	// Only log if tracing is enabled and the system is now initialized
	IF GPL_Base.TRACING_ENABLED AND_THEN GVL_System.RingBufferLog.P_RingBufferStatus.BaseStatus.Initialized THEN
		BaseStatus.LogEntry.Message								:= Message;
		BaseStatus.LogEntry.Severity							:= Severity;
		BaseStatus.LogEntry.RaiseAlarm							:= RaiseAlarm;
		BaseStatus.LogEntry.InstancePath						:= InstancePath;
		BaseStatus.LogEntry.TaskInfo.AdsPort					:= TwinCAT_SystemInfoVarList._TaskInfo[Tc2_System.GETCURTASKINDEXEX()].AdsPort;
		BaseStatus.LogEntry.TaskInfo.CycleCount					:= TwinCAT_SystemInfoVarList._TaskInfo[Tc2_System.GETCURTASKINDEXEX()].CycleCount;
		BaseStatus.LogEntry.TaskInfo.CycleTime					:= TwinCAT_SystemInfoVarList._TaskInfo[Tc2_System.GETCURTASKINDEXEX()].CycleTime;
		BaseStatus.LogEntry.TaskInfo.CycleTimeExceeded			:= TwinCAT_SystemInfoVarList._TaskInfo[Tc2_System.GETCURTASKINDEXEX()].CycleTimeExceeded;
		BaseStatus.LogEntry.TaskInfo.DcTaskTime					:= TwinCAT_SystemInfoVarList._TaskInfo[Tc2_System.GETCURTASKINDEXEX()].DcTaskTime;
		BaseStatus.LogEntry.TaskInfo.FirstCycle					:= TwinCAT_SystemInfoVarList._TaskInfo[Tc2_System.GETCURTASKINDEXEX()].FirstCycle;
//		BaseStatus.LogEntry.TaskInfo.InCallAfterOutputUpdate	:= TwinCAT_SystemInfoVarList._TaskInfo[Tc2_System.GETCURTASKINDEXEX()].InCallAfterOutputUpdate;
		BaseStatus.LogEntry.TaskInfo.LastExecTime				:= TwinCAT_SystemInfoVarList._TaskInfo[Tc2_System.GETCURTASKINDEXEX()].LastExecTime;
		BaseStatus.LogEntry.TaskInfo.ObjId						:= TwinCAT_SystemInfoVarList._TaskInfo[Tc2_System.GETCURTASKINDEXEX()].ObjId;
		BaseStatus.LogEntry.TaskInfo.Priority					:= TwinCAT_SystemInfoVarList._TaskInfo[Tc2_System.GETCURTASKINDEXEX()].Priority;
		BaseStatus.LogEntry.TaskInfo.RTViolation				:= TwinCAT_SystemInfoVarList._TaskInfo[Tc2_System.GETCURTASKINDEXEX()].RTViolation;
		BaseStatus.LogEntry.TaskInfo.TaskName					:= TwinCAT_SystemInfoVarList._TaskInfo[Tc2_System.GETCURTASKINDEXEX()].TaskName;
		GVL_System.RingBufferLog.AddObject(RefObject := BaseStatus.LogEntry);

		// Verify the entry was added successfully
		IF NOT GVL_System.RingBufferLog.P_ObjectWasAdded THEN
			// AddObject failed - buffer may be full or corrupted
			// Cannot use logging system to report this (would cause recursion)
			// Silently fail - the LogDequeue error handling will detect buffer issues
		ELSE
			// Successfully added - clear the flag
			GVL_System.RingBufferLog.ClearStatusFlagAdded();
		END_IF
	END_IF
END_IF

// Clear re-entry guard before exiting
GVL_System.InReentry_Logging := FALSE;
END_METHOD

END_FUNCTION_BLOCK

// Base/I_BaseStatic
INTERFACE I_BaseStatic EXTENDS __SYSTEM.IQueryInterface

PROPERTY Busy : BOOL
GET
END_GET
END_PROPERTY

PROPERTY Error : BOOL
GET
END_GET
END_PROPERTY

PROPERTY ErrorID : UDINT
GET
END_GET
END_PROPERTY

METHOD Initialize : BOOL
VAR_INPUT
END_VAR
END_METHOD

PROPERTY P_BaseConfiguration : REFERENCE TO ST_BaseConfiguration
GET
END_GET
END_PROPERTY

PROPERTY P_BaseStatus : REFERENCE TO ST_BaseStatus
GET
END_GET
END_PROPERTY

METHOD TraceWithSeverity
VAR_INPUT
	Message		: T_MaxString;
	Severity	: Global.TcEventSeverity;
	RaiseAlarm	: BOOL := FALSE;
END_VAR
END_METHOD

END_INTERFACE

// Base/I_BaseCyclic
INTERFACE I_BaseCyclic EXTENDS I_BaseStatic

METHOD CyclicLogic
END_METHOD

PROPERTY Initialized : BOOL
GET
END_GET
END_PROPERTY

END_INTERFACE

// Command/ITFs/I_Command
INTERFACE I_Command EXTENDS I_BaseCyclic

METHOD Abort : I_Command
END_METHOD

METHOD Cancel : I_Command
END_METHOD

METHOD Complete : I_Command
END_METHOD

METHOD Execute : I_Command
END_METHOD

METHOD InjectConfigurations
VAR_INPUT
    iComponent					: I_ComponentFull;
    iCommandConfiguration 		: I_CommandConfiguration;
    iPermIntlkConfiguration   	: I_PermIntlkConfiguration;
END_VAR
END_METHOD

PROPERTY P_CommandStatus : REFERENCE TO ST_CommandStatus
GET
END_GET
END_PROPERTY

METHOD Pause : I_Command
END_METHOD

METHOD Queue : I_Command
END_METHOD

METHOD Reset : I_Command
END_METHOD

METHOD Resume : I_Command
END_METHOD

METHOD Validate : I_Command
END_METHOD

END_INTERFACE

// Component/ITFs/I_ComponentFull
INTERFACE I_ComponentFull EXTENDS I_ComponentBase

METHOD DequeueCommand : BOOL
VAR_INPUT
	CmdIndex	: DINT;
END_VAR
END_METHOD

METHOD EnqueueCommand
VAR_INPUT
	CmdIndex	: DINT;
END_VAR
END_METHOD

{warning 'Add method implementation or delete method to use base implementation'}
METHOD ExecuteCommand : I_ComponentFull
VAR_INPUT
	CmdIndex	: DINT;
END_VAR
END_METHOD

METHOD PUBLIC GetIndexByPOUName : UINT
VAR_INPUT
	NameIn : T_MaxString;
END_VAR
END_METHOD

{warning 'Add method implementation or delete method to use base implementation'}
METHOD HMICommunication
END_METHOD

METHOD InjectCommandQueue
VAR_INPUT
	iCommandQueue : I_RingBufferICmd;
END_VAR
END_METHOD

PROPERTY P_CommandQueue : I_RingBufferICmd
GET
END_GET
END_PROPERTY

{warning 'Add property implementation or delete property to use base implementation'}
PROPERTY P_ComponentConfiguration : REFERENCE TO ST_ComponentConfiguration
GET
END_GET
END_PROPERTY

{warning 'Add property implementation or delete property to use base implementation'}
PROPERTY P_ComponentStatus : REFERENCE TO ST_ComponentStatus
GET
END_GET
END_PROPERTY

METHOD ResetAllCommands : E_CommandResult
END_METHOD

END_INTERFACE

// Component/ITFs/I_ComponentBase
INTERFACE I_ComponentBase EXTENDS I_BaseCyclic

METHOD InjectSystemInterfaces
VAR_INPUT
	SystemPermIntlk				: I_PermIntlk;
	ControlMode					: I_ControlMode;
END_VAR
END_METHOD

METHOD Reset : E_CommandResult
END_METHOD

END_INTERFACE

// PermIntlk/ITFs/I_PermIntlk
INTERFACE I_PermIntlk EXTENDS I_BaseCyclic

METHOD Evaluate : I_PermIntlk
END_METHOD

METHOD InjectPermIntlkConfiguration
VAR_INPUT
    iPermIntlkCfg 	: I_PermIntlkConfiguration;
END_VAR
END_METHOD

{attribute 'monitoring' := 'call'}
PROPERTY P_OK : BOOL
GET
END_GET
END_PROPERTY

PROPERTY P_PermIntlkStatus : REFERENCE TO ST_PermIntlkStatus
GET
END_GET
END_PROPERTY

END_INTERFACE

// PermIntlk/ITFs/I_PermIntlkConfiguration
INTERFACE I_PermIntlkConfiguration EXTENDS I_BaseStatic

PROPERTY P_PermIntlkConfiguration : REFERENCE TO ST_PermIntlkConfiguration
GET
END_GET
END_PROPERTY

END_INTERFACE

// ControlMode/ITFs/I_ControlMode
INTERFACE I_ControlMode EXTENDS I_BaseCyclic

METHOD ChangeMode : I_ControlMode
VAR_INPUT
	DesiredMode	: DINT;
END_VAR
END_METHOD

PROPERTY P_ControlMode : DINT
GET
END_GET
END_PROPERTY

END_INTERFACE

// RingBuffer/ITFs/I_RingBufferICmd
INTERFACE I_RingBufferICmd EXTENDS I_RingBufferBase

METHOD PUBLIC AddObject
VAR_INPUT
  RefObject           : REFERENCE TO ST_SystimeICmd;
END_VAR
VAR_OUTPUT
  Error               : BOOL;
END_VAR
END_METHOD

PROPERTY P_Buffer : REFERENCE TO ARRAY[GPL_RingBuffer.MIN_NUMBER_OBJECTS..GPL_RingBuffer.MAX_NUMBER_OBJECTS] OF ST_SystimeICmd;
GET
END_GET
END_PROPERTY

PROPERTY P_LastObjectPeeked : REFERENCE TO ST_SystimeICmd
GET
END_GET
END_PROPERTY

PROPERTY P_LastObjectRead : REFERENCE TO ST_SystimeICmd
GET
END_GET
END_PROPERTY

PROPERTY P_LastObjectRemoved : REFERENCE TO ST_SystimeICmd
GET
END_GET
END_PROPERTY

METHOD PUBLIC PeekObject : ST_SystimeICmd
END_METHOD

METHOD PUBLIC ReadObject : ST_SystimeICmd
VAR_OUTPUT
  Error : BOOL;
END_VAR
END_METHOD

END_INTERFACE

// RingBuffer/ITFs/I_RingBufferBase
INTERFACE I_RingBufferBase EXTENDS I_BaseStatic

METHOD ClearLastRemoved
END_METHOD

METHOD ClearStatusFlagAdded
END_METHOD

METHOD ClearStatusFlagPeeked
END_METHOD

METHOD ClearStatusFlagRead
END_METHOD

METHOD ClearStatusFlagRemoved
END_METHOD

PROPERTY P_ObjectWasAdded : REFERENCE TO BOOL
GET
END_GET
END_PROPERTY

PROPERTY P_ObjectWasPeeked : REFERENCE TO BOOL
GET
END_GET
END_PROPERTY

PROPERTY P_ObjectWasRead : REFERENCE TO BOOL
GET
END_GET
END_PROPERTY

PROPERTY P_ObjectWasRemoved : REFERENCE TO BOOL
GET
END_GET
END_PROPERTY

PROPERTY P_RingBufferStatus : REFERENCE TO ST_RingBufferStatus
GET
END_GET
END_PROPERTY

METHOD PUBLIC RemoveObject
VAR_OUTPUT
  Error              : BOOL;
END_VAR
END_METHOD

END_INTERFACE

// Command/ITFs/I_CommandConfiguration
INTERFACE I_CommandConfiguration EXTENDS I_BaseStatic

PROPERTY P_CommandConfiguration : REFERENCE TO ST_CommandConfiguration
GET
END_GET
END_PROPERTY

END_INTERFACE

// Command/ITFs/I_TestClock
INTERFACE I_TestClock

METHOD SetElapsedTime
VAR_INPUT
	DesiredET : LTIME;
END_VAR
END_METHOD

END_INTERFACE

// Command/ITFs/I_Timer
INTERFACE I_Timer EXTENDS __SYSTEM.IQueryInterface

PROPERTY P_ElapsedTime : TIME
GET
END_GET
END_PROPERTY

PROPERTY P_IsElapsed : BOOL
GET
END_GET
END_PROPERTY

METHOD ResetTimer
VAR_INPUT
END_VAR
END_METHOD

METHOD StartTimer
VAR_INPUT
END_VAR
END_METHOD

METHOD StopTimer
VAR_INPUT
END_VAR
END_METHOD

END_INTERFACE

// Command/POUs/FB_Command
{attribute 'no_explicit_call' := 'do not call this POU directly'}
{attribute 'enable_dynamic_creation'}
FUNCTION_BLOCK FB_Command EXTENDS FB_BaseCyclic IMPLEMENTS I_Command, I_CommandConfiguration
VAR
	iCommandInternal			: I_Command := THIS^;
	
 	_iComponent					: I_ComponentFull; // External Dependency
	_iCommandConfiguration		: I_CommandConfiguration; // External Dependency
	_iPermIntlkConfiguration	: I_PermIntlkConfiguration; // External Dependency
	
	LocalCommandConfiguration	: ST_CommandConfiguration := (CommandDescription := 'Missing Command Configuration Interface Reference'); //Local Reference Fallback
	LocalPermIntlkConfiguration	: ST_PermIntlkConfiguration; //Local Reference Fallback

 	fbPermIntlk					: FB_PermIntlkCommand;
	iPermIntlk					: I_PermIntlk := fbPermIntlk;
	
	fbCmdElapsedTime			: FB_CommandElapsedTimer;
	iTimer						: I_Timer := fbCmdElapsedTime;
	
	CommandStatus				: ST_CommandStatus;
	PreviousCommandStatus		: ST_CommandStatus;

	// Auto-reset timing for test compatibility
	CompleteStateCycles						: DINT := 0;
END_VAR

METHOD Abort : I_Command
// Guard condition derived from truth table
// B AND (E OR TO OR (PIC AND AID AND NOT ILK))
// Check external dependencies - only component required for queue operations
// Other dependencies are optional for basic abortion
IF (_iComponent = 0) THEN
	// Only log warning if we have a valid command configuration to read logging settings from
	IF (_iCommandConfiguration <> 0) THEN
		IF __ISVALIDREF(_iCommandConfiguration.P_CommandConfiguration.BaseConfiguration) THEN
			IF _iCommandConfiguration.P_CommandConfiguration.BaseConfiguration.LogTraceConfiguration.What.xLogToEventLogger THEN
				TraceWithSeverity(Message := 'Warning: Missing I_Component external dependency in Abort method - queue operations unavailable', Severity := Global.TcEventSeverity.Warning);
			END_IF
		END_IF
	END_IF
END_IF

// Abort should be available for any command that needs to be stopped or is active
IF SUPER^.BaseStatus.Initialized THEN

// Abort behavior depends on current state
CASE CommandStatus.StepState OF
    E_CommandState.Execute, E_CommandState.Monitor:
        // Abort executing or monitoring command
        _AbortCommand();
        IF (_iCommandConfiguration <> 0) THEN
            IF __ISVALIDREF(_iCommandConfiguration.P_CommandConfiguration.BaseConfiguration) THEN
                IF _iCommandConfiguration.P_CommandConfiguration.BaseConfiguration.LogTraceConfiguration.What.xLogToEventLogger THEN
                    TraceWithSeverity(Message := 'Command aborted during execution', Severity := Global.TcEventSeverity.Info);
                END_IF
            END_IF
        ELSE
            // WARNING: Event logging disabled - configuration interface is null
            TraceWithSeverity(Message := 'WARNING: _iCommandConfiguration is null in Abort - command aborted during execution logging disabled', Severity := Global.TcEventSeverity.Warning);
        END_IF

    E_CommandState.Idle:
        // Check if queued (by result) and remove from queue if present
        IF CommandStatus.Result = E_CommandResult.Accepted THEN // Queued commands have Accepted result
            IF _iComponent <> 0 THEN
                _iComponent.P_CommandQueue.PeekObject(); // peek each
                IF iCommandInternal = _iComponent.P_CommandQueue.P_LastObjectPeeked.iCmd THEN
                    _iComponent.P_CommandQueue.RemoveObject(); // find and remove specific instance
                END_IF
            END_IF
            IF (_iCommandConfiguration <> 0) THEN
                IF __ISVALIDREF(_iCommandConfiguration.P_CommandConfiguration.BaseConfiguration) THEN
                    IF _iCommandConfiguration.P_CommandConfiguration.BaseConfiguration.LogTraceConfiguration.What.xLogToEventLogger THEN
                        TraceWithSeverity(Message := 'Queued command aborted and removed from queue', Severity := Global.TcEventSeverity.Info);
                    END_IF
                END_IF
            ELSE
                // WARNING: Event logging disabled - configuration interface is null
                TraceWithSeverity(Message := 'WARNING: _iCommandConfiguration is null in Abort - queued command aborted and removed from queue logging disabled', Severity := Global.TcEventSeverity.Warning);
            END_IF
        ELSE
            IF (_iCommandConfiguration <> 0) THEN
                IF __ISVALIDREF(_iCommandConfiguration.P_CommandConfiguration.BaseConfiguration) THEN
                    IF _iCommandConfiguration.P_CommandConfiguration.BaseConfiguration.LogTraceConfiguration.What.xLogToEventLogger THEN
                        TraceWithSeverity(Message := 'Idle command marked as aborted', Severity := Global.TcEventSeverity.Info);
                    END_IF
                END_IF
            ELSE
                // WARNING: Event logging disabled - configuration interface is null
                TraceWithSeverity(Message := 'WARNING: _iCommandConfiguration is null in Abort - idle command marked as aborted logging disabled', Severity := Global.TcEventSeverity.Warning);
            END_IF
        END_IF
CommandStatus.Result := E_CommandResult.Aborted;

    E_CommandState.Paused:
        // Abort paused command
        _AbortCommand();
		IF (_iCommandConfiguration <> 0) THEN
			IF __ISVALIDREF(_iCommandConfiguration.P_CommandConfiguration.BaseConfiguration) THEN
				IF _iCommandConfiguration.P_CommandConfiguration.BaseConfiguration.LogTraceConfiguration.What.xLogToEventLogger THEN
					TraceWithSeverity(Message := 'Paused command aborted', Severity := Global.TcEventSeverity.Info);
				END_IF
			END_IF
		ELSE
			// WARNING: Event logging disabled - configuration interface is null
			TraceWithSeverity(Message := 'WARNING: _iCommandConfiguration is null in Abort - paused command aborted logging disabled', Severity := Global.TcEventSeverity.Warning);
		END_IF

    E_CommandState.Complete:
        // Policy: Abort-after-complete should not overwrite terminal results
        IF (_iCommandConfiguration <> 0) THEN
            IF __ISVALIDREF(_iCommandConfiguration.P_CommandConfiguration.BaseConfiguration) THEN
                IF _iCommandConfiguration.P_CommandConfiguration.BaseConfiguration.LogTraceConfiguration.What.xLogToEventLogger THEN
                    TraceWithSeverity(Message := 'Abort ignored - completed command preserves terminal result', Severity := Global.TcEventSeverity.Warning);
                END_IF
            END_IF
        ELSE
            // WARNING: Event logging disabled - configuration interface is null
            TraceWithSeverity(Message := 'WARNING: _iCommandConfiguration is null in Abort - abort ignored for completed command logging disabled', Severity := Global.TcEventSeverity.Warning);
        END_IF
        // Do not change CommandStatus.Result to preserve Ok/RequestTimeout/InterlockLost etc.
END_CASE

ELSE
    // FB not initialized - cannot safely abort
    IF (_iCommandConfiguration <> 0) THEN
        IF __ISVALIDREF(_iCommandConfiguration.P_CommandConfiguration.BaseConfiguration) THEN
            IF _iCommandConfiguration.P_CommandConfiguration.BaseConfiguration.LogTraceConfiguration.What.xLogToEventLogger THEN
                TraceWithSeverity(Message := 'Cannot abort - FB_Command not initialized', Severity := Global.TcEventSeverity.Error);
            END_IF
        END_IF
    ELSE
        // WARNING: Event logging disabled - configuration interface is null
        TraceWithSeverity(Message := 'WARNING: _iCommandConfiguration is null in Abort - FB_Command not initialized logging disabled', Severity := Global.TcEventSeverity.Warning);
    END_IF
END_IF

Abort := THIS^;
END_METHOD

METHOD Cancel : I_Command
// Guard condition derived from truth table
// NOT B AND NOT E AND NOT D
// Check external dependencies - only component required for queue operations
// Other dependencies are optional for basic cancellation
IF (_iComponent = 0) THEN
	// Only log warning if we have a valid command configuration to read logging settings from
	IF (_iCommandConfiguration <> 0) THEN
		IF __ISVALIDREF(_iCommandConfiguration.P_CommandConfiguration.BaseConfiguration) THEN
			IF _iCommandConfiguration.P_CommandConfiguration.BaseConfiguration.LogTraceConfiguration.What.xLogToEventLogger THEN
				TraceWithSeverity(Message := 'Warning: Missing I_Component external dependency in Cancel method - queue operations unavailable', Severity := Global.TcEventSeverity.Warning);
			END_IF
		END_IF
	ELSE
		// WARNING: Event logging disabled - configuration interface is null
		TraceWithSeverity(Message := 'WARNING: _iCommandConfiguration is null in Cancel - missing I_Component dependency logging disabled', Severity := Global.TcEventSeverity.Warning);
	END_IF
END_IF

// Cancel behavior depends on current state, not on Done flag
// Allow cancel for idle and paused states regardless of Done status
CASE CommandStatus.StepState OF
    E_CommandState.Idle:
        // Check if queued (by result) and remove from queue if present
        IF CommandStatus.Result = E_CommandResult.Accepted THEN // Queued commands have Accepted result
            IF _iComponent <> 0 THEN
                _iComponent.P_CommandQueue.PeekObject(); // peek each
                IF iCommandInternal = _iComponent.P_CommandQueue.P_LastObjectPeeked.iCmd THEN
                    _iComponent.P_CommandQueue.RemoveObject(); // find and remove specific instance
                END_IF
            END_IF
            IF (_iCommandConfiguration <> 0) THEN
                IF __ISVALIDREF(_iCommandConfiguration.P_CommandConfiguration.BaseConfiguration) THEN
                    IF _iCommandConfiguration.P_CommandConfiguration.BaseConfiguration.LogTraceConfiguration.What.xLogToEventLogger THEN
                        TraceWithSeverity(Message := 'Queued command cancelled and removed from queue', Severity := Global.TcEventSeverity.Info);
                    END_IF
                END_IF
            ELSE
                // WARNING: Event logging disabled - configuration interface is null
                TraceWithSeverity(Message := 'WARNING: _iCommandConfiguration is null in Cancel - queued command cancelled logging disabled', Severity := Global.TcEventSeverity.Warning);
            END_IF
        ELSE
            // Regular idle command - still set cancelled result
            IF (_iCommandConfiguration <> 0) THEN
                IF __ISVALIDREF(_iCommandConfiguration.P_CommandConfiguration.BaseConfiguration) THEN
                    IF _iCommandConfiguration.P_CommandConfiguration.BaseConfiguration.LogTraceConfiguration.What.xLogToEventLogger THEN
                        TraceWithSeverity(Message := 'Idle command cancelled', Severity := Global.TcEventSeverity.Info);
                    END_IF
                END_IF
            ELSE
                // WARNING: Event logging disabled - configuration interface is null
                TraceWithSeverity(Message := 'WARNING: _iCommandConfiguration is null in Cancel - idle command cancelled logging disabled', Severity := Global.TcEventSeverity.Warning);
            END_IF
        END_IF
        // Set cancelled result for any idle command, stay in Idle state
        CommandStatus.Result := E_CommandResult.Cancelled;
                IF __ISVALIDREF(CommandStatus.BaseStatus) THEN
            CommandStatus.BaseStatus.Error := FALSE;  // Cancelled is not an error
                    ELSE
            TraceWithSeverity(Message := 'Command Base Reference Data Structure not present - see _InitializeReferences', Severity := Global.TcEventSeverity.Error);
        END_IF
        
    E_CommandState.Execute, E_CommandState.Monitor:
        // Policy: Cancel should not change results while busy - do nothing
        IF (_iCommandConfiguration <> 0) THEN
            IF __ISVALIDREF(_iCommandConfiguration.P_CommandConfiguration.BaseConfiguration) THEN
                IF _iCommandConfiguration.P_CommandConfiguration.BaseConfiguration.LogTraceConfiguration.What.xLogToEventLogger THEN
                    TraceWithSeverity(Message := 'Cancel rejected - command is executing, use Abort instead', Severity := Global.TcEventSeverity.Warning);
                END_IF
            END_IF
        ELSE
            // WARNING: Event logging disabled - configuration interface is null
            TraceWithSeverity(Message := 'WARNING: _iCommandConfiguration is null in Cancel - cancel rejected (executing) logging disabled', Severity := Global.TcEventSeverity.Warning);
        END_IF
        // Do not change CommandStatus.Result
        
    E_CommandState.Paused:
        // Policy: Cancel should not change results while paused/busy - do nothing
        IF (_iCommandConfiguration <> 0) THEN
            IF __ISVALIDREF(_iCommandConfiguration.P_CommandConfiguration.BaseConfiguration) THEN
                IF _iCommandConfiguration.P_CommandConfiguration.BaseConfiguration.LogTraceConfiguration.What.xLogToEventLogger THEN
                    TraceWithSeverity(Message := 'Cancel rejected - command is paused, use Abort instead', Severity := Global.TcEventSeverity.Warning);
                END_IF
            END_IF
        ELSE
            // WARNING: Event logging disabled - configuration interface is null
            TraceWithSeverity(Message := 'WARNING: _iCommandConfiguration is null in Cancel - cancel rejected (paused) logging disabled', Severity := Global.TcEventSeverity.Warning);
        END_IF
        // Do not change CommandStatus.Result

    E_CommandState.Complete:
        // Policy: Cancel should not change results while complete - do nothing
        IF (_iCommandConfiguration <> 0) THEN
            IF __ISVALIDREF(_iCommandConfiguration.P_CommandConfiguration.BaseConfiguration) THEN
                IF _iCommandConfiguration.P_CommandConfiguration.BaseConfiguration.LogTraceConfiguration.What.xLogToEventLogger THEN
                    TraceWithSeverity(Message := 'Cancel rejected - command is complete', Severity := Global.TcEventSeverity.Warning);
                END_IF
            END_IF
        ELSE
            // WARNING: Event logging disabled - configuration interface is null
            TraceWithSeverity(Message := 'WARNING: _iCommandConfiguration is null in Cancel - cancel rejected (complete) logging disabled', Severity := Global.TcEventSeverity.Warning);
        END_IF
        // Do not change CommandStatus.Result
END_CASE

Cancel := THIS^;
END_METHOD

METHOD Complete : I_Command
// Mark command as no longer busy when completion is triggered
// This allows the component to accept new commands immediately
IF CommandStatus.StepState = E_CommandState.Monitor THEN
    IF __ISVALIDREF(CommandStatus.BaseStatus) THEN
        CommandStatus.BaseStatus.Busy := FALSE;
            ELSE
        TraceWithSeverity(Message := 'Command Base Reference Data Structure not present - see _InitializeReferences', Severity := Global.TcEventSeverity.Error);
    END_IF
    // Stop the elapsed timer to prevent it from continuing to increment
    IF iTimer <> 0 THEN
        iTimer.StopTimer();
    END_IF
END_IF

Complete := THIS^;
END_METHOD

METHOD Execute : I_Command
// Critical check: Timer interface must be present for command execution
IF iTimer = 0 THEN
	TraceWithSeverity(
		Message := 'CRITICAL: Cannot execute command - timer interface not present! Timeout monitoring would not work!',
		Severity := Global.TcEventSeverity.Error
	);
	CommandStatus.Result := E_CommandResult.BadRequest;
	Execute := THIS^;
	RETURN;
END_IF

// Guard condition derived from truth table
// NOT B AND NOT E AND NOT D AND ILK AND NOT TO
// Check external dependencies - allow execution with minimal configuration for basic testing
IF (_iComponent = 0) THEN
	// Only log warning if we have a valid command configuration to read logging settings from
	IF (_iCommandConfiguration <> 0) THEN
		IF __ISVALIDREF(_iCommandConfiguration.P_CommandConfiguration.BaseConfiguration) THEN
			IF _iCommandConfiguration.P_CommandConfiguration.BaseConfiguration.LogTraceConfiguration.What.xLogToEventLogger THEN
				TraceWithSeverity(Message := 'Warning: Missing I_Component external dependency in Execute method - advanced features unavailable', Severity := Global.TcEventSeverity.Warning);
			END_IF
		END_IF
	END_IF
END_IF

// Check timeout condition safely
IF (_iCommandConfiguration <> 0) THEN
    IF CommandStatus.LastCommandElapsedTime >= TIME_TO_LTIME(_iCommandConfiguration.P_CommandConfiguration.TimeoutTime) THEN
        CommandStatus.Result := E_CommandResult.RequestTimeout;
                IF __ISVALIDREF(CommandStatus.BaseStatus) THEN
            CommandStatus.BaseStatus.Error := TRUE;  // Set error flag for timeout
                        CommandStatus.BaseStatus.Done := TRUE;  // Complete state always sets Done=TRUE (terminal state)
                    ELSE
            TraceWithSeverity(Message := 'Command Base Reference Data Structure not present - see _InitializeReferences', Severity := Global.TcEventSeverity.Error);
        END_IF
        IF __ISVALIDREF(_iCommandConfiguration.P_CommandConfiguration.BaseConfiguration) THEN
            IF _iCommandConfiguration.P_CommandConfiguration.BaseConfiguration.LogTraceConfiguration.What.xLogToEventLogger THEN
                TraceWithSeverity(Message := 'Command timeout exceeded in Execute method', Severity := Global.TcEventSeverity.Error);
            END_IF
        END_IF
    END_IF
ELSE
    // WARNING: Cannot check timeout without configuration - execution may proceed beyond timeout
    TraceWithSeverity(Message := 'WARNING: _iCommandConfiguration is null in Execute method - timeout check bypassed', Severity := Global.TcEventSeverity.Warning);
END_IF

// Enhanced guard conditions - prevent execution in terminal states
// Execute should only be allowed from clean Idle state
IF SUPER^.BaseStatus.Initialized AND 
   NOT CommandStatus.BaseStatus.Busy AND 
   NOT CommandStatus.BaseStatus.Done AND
   NOT CommandStatus.BaseStatus.Error THEN

// Execute behavior depends on current state
CASE CommandStatus.StepState OF
    E_CommandState.Idle:
        // Execute must validate before accepting - call Validate() internally
        _ValidateCommand();
        
        // Only proceed if validation was successful (Accepted)
        IF CommandStatus.Result = E_CommandResult.Accepted THEN
            
            // Optional trace
            IF (_iCommandConfiguration <> 0) THEN
                IF __ISVALIDREF(_iCommandConfiguration.P_CommandConfiguration.BaseConfiguration) THEN
                    IF _iCommandConfiguration.P_CommandConfiguration.BaseConfiguration.LogTraceConfiguration.When = E_LogTraceWhen.xRunCyclic AND_THEN
                       _iCommandConfiguration.P_CommandConfiguration.BaseConfiguration.LogTraceConfiguration.What.xLogToEventLogger THEN
                        _LogCommand();
                    END_IF
                END_IF
            ELSE
                // WARNING: Event logging disabled - configuration interface is null
                TraceWithSeverity(Message := 'WARNING: _iCommandConfiguration is null in Execute - optional trace logging disabled', Severity := Global.TcEventSeverity.Warning);
            END_IF
            
            // Set Busy flag to enable state transitions - validation already passed
            IF __ISVALIDREF(CommandStatus.BaseStatus) THEN
                CommandStatus.BaseStatus.Busy := TRUE;
                            ELSE
                TraceWithSeverity(Message := 'Command Base Reference Data Structure not present - see _InitializeReferences', Severity := Global.TcEventSeverity.Error);
            END_IF

            // Start the command timer to track elapsed time
            IF iTimer <> 0 THEN
                iTimer.StartTimer();
            END_IF
            // Keep Result as Accepted - CyclicLogic will drive state progression
        END_IF
        // If validation failed, Result already contains the failure reason (Forbidden, BadRequest, etc.)
        
    E_CommandState.Execute, E_CommandState.Monitor, E_CommandState.Complete:
        // Already executing, monitoring, or complete - cannot execute again
        // Complete is a terminal state - use Reset() to return to Idle for re-execution
        IF (_iCommandConfiguration <> 0) THEN
            IF __ISVALIDREF(_iCommandConfiguration.P_CommandConfiguration.BaseConfiguration) THEN
                IF _iCommandConfiguration.P_CommandConfiguration.BaseConfiguration.LogTraceConfiguration.What.xLogToEventLogger THEN
                    TraceWithSeverity(Message := 'Cannot execute - command already in progress or complete. Use Reset() first.', Severity := Global.TcEventSeverity.Warning);
                END_IF
            END_IF
        ELSE
            // WARNING: Event logging disabled - configuration interface is null
            TraceWithSeverity(Message := 'WARNING: _iCommandConfiguration is null in Execute - already in progress/complete logging disabled', Severity := Global.TcEventSeverity.Warning);
        END_IF

    E_CommandState.Paused:
        // Cannot execute from paused state - use Resume instead
        IF (_iCommandConfiguration <> 0) THEN
            IF __ISVALIDREF(_iCommandConfiguration.P_CommandConfiguration.BaseConfiguration) THEN
                IF _iCommandConfiguration.P_CommandConfiguration.BaseConfiguration.LogTraceConfiguration.What.xLogToEventLogger THEN
                    TraceWithSeverity(Message := 'Cannot execute - command is paused, use Resume instead', Severity := Global.TcEventSeverity.Warning);
                END_IF
            END_IF
        ELSE
            // WARNING: Event logging disabled - configuration interface is null
            TraceWithSeverity(Message := 'WARNING: _iCommandConfiguration is null in Execute - paused state logging disabled', Severity := Global.TcEventSeverity.Warning);
        END_IF
END_CASE

ELSE
	// Guard condition not met - command not initialized, busy, or in terminal state
	IF NOT SUPER^.BaseStatus.Initialized THEN
	    CommandStatus.Result := E_CommandResult.BadRequest;
	    	    IF __ISVALIDREF(CommandStatus.BaseStatus) THEN
	        CommandStatus.BaseStatus.Error := TRUE;  // Set error flag for bad request
	        	    ELSE
	        TraceWithSeverity(Message := 'Command Base Reference Data Structure not present - see _InitializeReferences', Severity := Global.TcEventSeverity.Error);
	    END_IF
	    IF (_iCommandConfiguration <> 0) THEN
	    	IF __ISVALIDREF(_iCommandConfiguration.P_CommandConfiguration.BaseConfiguration) THEN
	            IF _iCommandConfiguration.P_CommandConfiguration.BaseConfiguration.LogTraceConfiguration.What.xLogToEventLogger THEN
	                TraceWithSeverity(Message := 'Execute failed - command not initialized', Severity := Global.TcEventSeverity.Warning);
	            END_IF
	        END_IF
	    ELSE
	        // WARNING: Event logging disabled - configuration interface is null
	        TraceWithSeverity(Message := 'WARNING: _iCommandConfiguration is null in Execute - not initialized logging disabled', Severity := Global.TcEventSeverity.Warning);
	    END_IF
	ELSIF CommandStatus.BaseStatus.Busy THEN
	    CommandStatus.Result := E_CommandResult.Forbidden;
	    	    IF __ISVALIDREF(CommandStatus.BaseStatus) THEN
	        CommandStatus.BaseStatus.Error := TRUE;  // Set error flag for forbidden
	        	    ELSE
	        TraceWithSeverity(Message := 'Command Base Reference Data Structure not present - see _InitializeReferences', Severity := Global.TcEventSeverity.Error);
	    END_IF
	    IF (_iCommandConfiguration <> 0) THEN
	    	IF __ISVALIDREF(_iCommandConfiguration.P_CommandConfiguration.BaseConfiguration) THEN
	            IF _iCommandConfiguration.P_CommandConfiguration.BaseConfiguration.LogTraceConfiguration.What.xLogToEventLogger THEN
	                TraceWithSeverity(Message := 'Execute failed - command busy', Severity := Global.TcEventSeverity.Warning);
	            END_IF
	        END_IF
	    ELSE
	        // WARNING: Event logging disabled - configuration interface is null
	        TraceWithSeverity(Message := 'WARNING: _iCommandConfiguration is null in Execute - command busy logging disabled', Severity := Global.TcEventSeverity.Warning);
	    END_IF
	END_IF
END_IF

Execute := THIS^;
END_METHOD

METHOD InjectConfigurations
VAR_INPUT
    iComponent					: I_ComponentFull;
    iCommandConfiguration 		: I_CommandConfiguration;
    iPermIntlkConfiguration   	: I_PermIntlkConfiguration;
END_VAR
// Inject component interface (moved from FB_Init)
IF iComponent <> 0 THEN
	THIS^._iComponent := iComponent;
	IF NOT SUPER^.BaseStatus.LogTraceStatus.ComponentInterfaceInjectedShown THEN
		TraceWithSeverity(Message := 'FB_Command: Component interface injected successfully', Severity := Global.TcEventSeverity.Verbose);
		SUPER^.BaseStatus.LogTraceStatus.ComponentInterfaceInjectedShown := TRUE;
	END_IF
END_IF

// Inject configuration interfaces (allow null interfaces for testing)
// Null interfaces clear the stored reference to force fallback to local config
IF iCommandConfiguration <> 0 THEN
    _iCommandConfiguration := iCommandConfiguration;
    IF NOT SUPER^.BaseStatus.LogTraceStatus.CmdConfigInterfaceInjectedShown THEN
		TraceWithSeverity(Message := 'FB_Command: Command configuration interface injected successfully', Severity := Global.TcEventSeverity.Verbose);
		SUPER^.BaseStatus.LogTraceStatus.CmdConfigInterfaceInjectedShown := TRUE;
	END_IF
ELSE
    IF (_iCommandConfiguration <> 0) THEN
        IF __ISVALIDREF(_iCommandConfiguration.P_CommandConfiguration.BaseConfiguration) THEN
            IF _iCommandConfiguration.P_CommandConfiguration.BaseConfiguration.LogTraceConfiguration.What.xLogToEventLogger THEN
                TraceWithSeverity(Message := 'Null Command Configuration interface injected - clearing reference', Severity := Global.TcEventSeverity.Info);
            END_IF
        END_IF
    END_IF
    _iCommandConfiguration := 0; // Clear the reference
END_IF

IF iPermIntlkConfiguration <> 0 THEN
    _iPermIntlkConfiguration := iPermIntlkConfiguration;
    IF NOT SUPER^.BaseStatus.LogTraceStatus.PermIntlkConfigInjectedShown THEN
		TraceWithSeverity(Message := 'FB_Command: PermIntlk configuration interface injected successfully', Severity := Global.TcEventSeverity.Verbose);
		SUPER^.BaseStatus.LogTraceStatus.PermIntlkConfigInjectedShown := TRUE;
	END_IF
ELSE
    IF (_iCommandConfiguration <> 0) THEN
        IF __ISVALIDREF(_iCommandConfiguration.P_CommandConfiguration.BaseConfiguration) THEN
            IF _iCommandConfiguration.P_CommandConfiguration.BaseConfiguration.LogTraceConfiguration.What.xLogToEventLogger THEN
                TraceWithSeverity(Message := 'Null PermIntlk Configuration interface injected - clearing reference', Severity := Global.TcEventSeverity.Info);
            END_IF
        END_IF
    END_IF
    _iPermIntlkConfiguration := 0; // Clear the reference
END_IF

// Only inject to child objects if interfaces are valid
IF iCommandConfiguration <> 0 THEN
    fbPermIntlk.InjectCommandConfiguration(iCommandCfg := iCommandConfiguration);
    fbCmdElapsedTime.InjectConfiguration(iCommand := THIS^, iCommandConfiguration := iCommandConfiguration);
    IF NOT SUPER^.BaseStatus.LogTraceStatus.ConfigsInjectedToChildrenShown THEN
		TraceWithSeverity(Message := 'FB_Command: Configurations injected to child objects (fbPermIntlk, fbCmdElapsedTime)', Severity := Global.TcEventSeverity.Verbose);
		SUPER^.BaseStatus.LogTraceStatus.ConfigsInjectedToChildrenShown := TRUE;
	END_IF
END_IF

IF iPermIntlkConfiguration <> 0 THEN
    fbPermIntlk.InjectPermIntlkConfiguration(iPermIntlkCfg := iPermIntlkConfiguration);
    // Ensure permissive interface is properly initialized
    fbPermIntlk.Initialize();
    IF NOT SUPER^.BaseStatus.LogTraceStatus.PermIntlkInitializedShown THEN
		TraceWithSeverity(Message := 'FB_Command: PermIntlk configuration injected and initialized in fbPermIntlk', Severity := Global.TcEventSeverity.Verbose);
		SUPER^.BaseStatus.LogTraceStatus.PermIntlkInitializedShown := TRUE;
	END_IF
END_IF

// Initialize the command after dependency injection
// This ensures all interfaces are available before initialization
THIS^.Initialize();

// Set BadRequest result if required configurations are missing (fail-closed policy)
IF (_iCommandConfiguration = 0) OR (_iPermIntlkConfiguration = 0) THEN
    CommandStatus.Result := E_CommandResult.BadRequest;
        IF __ISVALIDREF(CommandStatus.BaseStatus) THEN
        CommandStatus.BaseStatus.Error := TRUE;
            ELSE
        TraceWithSeverity(Message := 'Command Base Reference Data Structure not present - see _InitializeReferences', Severity := Global.TcEventSeverity.Error);
    END_IF
END_IF;
END_METHOD

PROPERTY P_CommandStatus : REFERENCE TO ST_CommandStatus
GET
P_CommandStatus REF= _ResolveCommandStatus();
END_GET
END_PROPERTY

METHOD Pause : I_Command
// Guard condition derived from truth table
// B AND NOT E AND NOT D
// Check external dependencies - allow basic pause functionality with warnings
IF (_iComponent = 0) THEN
	// Only log warning if we have a valid command configuration to read logging settings from
	IF (_iCommandConfiguration <> 0) THEN
		IF __ISVALIDREF(_iCommandConfiguration.P_CommandConfiguration) THEN
			IF __ISVALIDREF(_iCommandConfiguration.P_CommandConfiguration.BaseConfiguration) THEN
				IF _iCommandConfiguration.P_CommandConfiguration.BaseConfiguration.LogTraceConfiguration.What.xLogToEventLogger THEN
					TraceWithSeverity(Message := 'Warning: Missing I_Component external dependency in Pause method', Severity := Global.TcEventSeverity.Warning);
				END_IF
			END_IF
		END_IF
	ELSE
		// WARNING: Event logging disabled - configuration interface is null
		TraceWithSeverity(Message := 'WARNING: _iCommandConfiguration is null in Pause - missing I_Component dependency logging disabled', Severity := Global.TcEventSeverity.Warning);
	END_IF
END_IF

IF CommandStatus.BaseStatus.Busy AND 
   NOT CommandStatus.BaseStatus.Error AND 
   NOT CommandStatus.BaseStatus.Done THEN

// Pause behavior depends on current state
CASE CommandStatus.StepState OF
    E_CommandState.Execute, E_CommandState.Monitor:
        // Pause executing or monitoring command
        CommandStatus.StepState := E_CommandState.Paused;
                // Keep Busy = TRUE while paused (paused commands are active but suspended)
        // CommandStatus.BaseStatus.Busy remains TRUE
        IF (_iCommandConfiguration <> 0) THEN
            IF __ISVALIDREF(_iCommandConfiguration.P_CommandConfiguration.BaseConfiguration) THEN
                IF _iCommandConfiguration.P_CommandConfiguration.BaseConfiguration.LogTraceConfiguration.What.xLogToEventLogger THEN
                    TraceWithSeverity(Message := 'Command paused during execution', Severity := Global.TcEventSeverity.Info);
                END_IF
            END_IF
        ELSE
            // WARNING: Event logging disabled - configuration interface is null
            TraceWithSeverity(Message := 'WARNING: _iCommandConfiguration is null in Pause - command paused during execution logging disabled', Severity := Global.TcEventSeverity.Warning);
        END_IF
        
    // Note: Queued commands are now Idle with Accepted result
        
    E_CommandState.Idle:
        // Cannot pause idle command
        IF (_iCommandConfiguration <> 0) THEN
            IF __ISVALIDREF(_iCommandConfiguration.P_CommandConfiguration.BaseConfiguration) THEN
                IF _iCommandConfiguration.P_CommandConfiguration.BaseConfiguration.LogTraceConfiguration.What.xLogToEventLogger THEN
                    TraceWithSeverity(Message := 'Cannot pause idle command', Severity := Global.TcEventSeverity.Warning);
                END_IF
            END_IF
        ELSE
            // WARNING: Event logging disabled - configuration interface is null
            TraceWithSeverity(Message := 'WARNING: _iCommandConfiguration is null in Pause - cannot pause idle command logging disabled', Severity := Global.TcEventSeverity.Warning);
        END_IF
        
    E_CommandState.Paused:
        // Already paused
        IF (_iCommandConfiguration <> 0) THEN
            IF __ISVALIDREF(_iCommandConfiguration.P_CommandConfiguration.BaseConfiguration) THEN
                IF _iCommandConfiguration.P_CommandConfiguration.BaseConfiguration.LogTraceConfiguration.What.xLogToEventLogger THEN
                    TraceWithSeverity(Message := 'Command is already paused', Severity := Global.TcEventSeverity.Info);
                END_IF
            END_IF
        ELSE
            // WARNING: Event logging disabled - configuration interface is null
            TraceWithSeverity(Message := 'WARNING: _iCommandConfiguration is null in Pause - already paused logging disabled', Severity := Global.TcEventSeverity.Warning);
        END_IF
        
    E_CommandState.Complete:
        // Cannot pause completed command
        IF (_iCommandConfiguration <> 0) THEN
            IF __ISVALIDREF(_iCommandConfiguration.P_CommandConfiguration.BaseConfiguration) THEN
                IF _iCommandConfiguration.P_CommandConfiguration.BaseConfiguration.LogTraceConfiguration.What.xLogToEventLogger THEN
                    TraceWithSeverity(Message := 'Cannot pause completed command', Severity := Global.TcEventSeverity.Warning);
                END_IF
            END_IF
        ELSE
            // WARNING: Event logging disabled - configuration interface is null
            TraceWithSeverity(Message := 'WARNING: _iCommandConfiguration is null in Pause - cannot pause completed command logging disabled', Severity := Global.TcEventSeverity.Warning);
        END_IF
END_CASE

ELSE
	// Guard condition not met - pause not allowed
	IF (_iCommandConfiguration <> 0) THEN
		IF __ISVALIDREF(_iCommandConfiguration.P_CommandConfiguration.BaseConfiguration) THEN
			IF _iCommandConfiguration.P_CommandConfiguration.BaseConfiguration.LogTraceConfiguration.What.xLogToEventLogger THEN
				TraceWithSeverity(Message := 'Pause guard condition not met', Severity := Global.TcEventSeverity.Warning);
			END_IF
		END_IF
	ELSE
		// WARNING: Event logging disabled - configuration interface is null
		TraceWithSeverity(Message := 'WARNING: _iCommandConfiguration is null in Pause - guard condition not met logging disabled', Severity := Global.TcEventSeverity.Warning);
	END_IF
END_IF

Pause := THIS^;
END_METHOD

METHOD Queue : I_Command
// Guard condition derived from truth table
// NOT B AND NOT E
// Check external dependencies
IF (_iComponent = 0) THEN
	// Only log warning if we have a valid command configuration to read logging settings from
	IF (_iCommandConfiguration <> 0) THEN
		IF __ISVALIDREF(_iCommandConfiguration.P_CommandConfiguration) THEN
			IF __ISVALIDREF(_iCommandConfiguration.P_CommandConfiguration.BaseConfiguration) THEN
				IF _iCommandConfiguration.P_CommandConfiguration.BaseConfiguration.LogTraceConfiguration.What.xLogToEventLogger THEN
					TraceWithSeverity(Message := 'Missing I_Component external dependency in Queue method', Severity := Global.TcEventSeverity.Error);
				END_IF
			END_IF
		END_IF
	ELSE
		// WARNING: Event logging disabled - configuration interface is null
		TraceWithSeverity(Message := 'WARNING: _iCommandConfiguration is null in Queue - missing I_Component dependency logging disabled', Severity := Global.TcEventSeverity.Warning);
	END_IF
	RETURN;
END_IF
IF (_iCommandConfiguration = 0) THEN
	// CRITICAL: Cannot queue without command configuration
	TraceWithSeverity(Message := 'CRITICAL: _iCommandConfiguration is null in Queue method - queue operation rejected', Severity := Global.TcEventSeverity.Error);
	RETURN;
END_IF
IF (_iPermIntlkConfiguration = 0) THEN
	// Log using the valid command configuration we already verified exists
	IF __ISVALIDREF(_iCommandConfiguration.P_CommandConfiguration) THEN
		IF __ISVALIDREF(_iCommandConfiguration.P_CommandConfiguration.BaseConfiguration) THEN
			IF _iCommandConfiguration.P_CommandConfiguration.BaseConfiguration.LogTraceConfiguration.What.xLogToEventLogger THEN
				TraceWithSeverity(Message := 'Missing I_PermIntlkConfiguration external dependency in Queue method', Severity := Global.TcEventSeverity.Error);
			END_IF
		END_IF
	END_IF
	RETURN;
END_IF

IF NOT CommandStatus.BaseStatus.Busy AND 
   NOT CommandStatus.BaseStatus.Error THEN

// Queue behavior depends on current state
CASE CommandStatus.StepState OF
    E_CommandState.Idle:
        // Check if already queued by looking at result
        IF CommandStatus.Result = E_CommandResult.Accepted THEN
            IF (_iCommandConfiguration <> 0) THEN
                IF __ISVALIDREF(_iCommandConfiguration.P_CommandConfiguration.BaseConfiguration) THEN
                    IF _iCommandConfiguration.P_CommandConfiguration.BaseConfiguration.LogTraceConfiguration.What.xLogToEventLogger THEN
                        TraceWithSeverity(Message := 'Command is already queued', Severity := Global.TcEventSeverity.Info);
                    END_IF
                END_IF
            ELSE
                // WARNING: Event logging disabled - configuration interface is null
                TraceWithSeverity(Message := 'WARNING: _iCommandConfiguration is null in Queue - already queued logging disabled', Severity := Global.TcEventSeverity.Warning);
            END_IF
        ELSE
            // Queue idle command
            IF _iComponent <> 0 THEN
                IF _iCommandConfiguration <> 0 THEN
                    IF __ISVALIDREF(_iCommandConfiguration.P_CommandConfiguration) THEN
                        _iComponent.EnqueueCommand(CmdIndex := _iCommandConfiguration.P_CommandConfiguration.CommandIndex);
                        CommandStatus.Result := E_CommandResult.Accepted; // Queued = Idle state with Accepted result
                                                IF (_iCommandConfiguration <> 0) THEN
                            IF __ISVALIDREF(_iCommandConfiguration.P_CommandConfiguration.BaseConfiguration) THEN
                                IF _iCommandConfiguration.P_CommandConfiguration.BaseConfiguration.LogTraceConfiguration.What.xLogToEventLogger THEN
                                    TraceWithSeverity(Message := 'Command queued successfully', Severity := Global.TcEventSeverity.Info);
                                END_IF
                            END_IF
                        ELSE
                            // WARNING: Event logging disabled - configuration interface is null
                            TraceWithSeverity(Message := 'WARNING: _iCommandConfiguration is null in Queue - command queued successfully logging disabled', Severity := Global.TcEventSeverity.Warning);
                        END_IF
                    ELSE
                        IF (_iCommandConfiguration <> 0) THEN
                            IF __ISVALIDREF(_iCommandConfiguration.P_CommandConfiguration.BaseConfiguration) THEN
                                IF _iCommandConfiguration.P_CommandConfiguration.BaseConfiguration.LogTraceConfiguration.What.xLogToEventLogger THEN
                                    TraceWithSeverity(Message := 'Cannot queue - P_CommandConfiguration reference invalid', Severity := Global.TcEventSeverity.Error);
                                END_IF
                            END_IF
                        ELSE
                            // WARNING: Event logging disabled - configuration interface is null
                            TraceWithSeverity(Message := 'WARNING: _iCommandConfiguration is null in Queue - invalid config reference logging disabled', Severity := Global.TcEventSeverity.Warning);
                        END_IF
                        RETURN;
                    END_IF
                ELSE
                    IF (_iCommandConfiguration <> 0) THEN
                        IF __ISVALIDREF(_iCommandConfiguration.P_CommandConfiguration.BaseConfiguration) THEN
                            IF _iCommandConfiguration.P_CommandConfiguration.BaseConfiguration.LogTraceConfiguration.What.xLogToEventLogger THEN
                                TraceWithSeverity(Message := 'Cannot queue - missing command configuration', Severity := Global.TcEventSeverity.Error);
                            END_IF
                        END_IF
                    ELSE
                        // WARNING: Event logging disabled - configuration interface is null
                        TraceWithSeverity(Message := 'WARNING: _iCommandConfiguration is null in Queue - missing command configuration logging disabled', Severity := Global.TcEventSeverity.Warning);
                    END_IF
                    RETURN;
                END_IF
            ELSE
                IF (_iCommandConfiguration <> 0) THEN
                    IF __ISVALIDREF(_iCommandConfiguration.P_CommandConfiguration.BaseConfiguration) THEN
                        IF _iCommandConfiguration.P_CommandConfiguration.BaseConfiguration.LogTraceConfiguration.What.xLogToEventLogger THEN
                            TraceWithSeverity(Message := 'Cannot queue - missing component interface', Severity := Global.TcEventSeverity.Error);
                        END_IF
                    END_IF
                ELSE
                    // WARNING: Event logging disabled - configuration interface is null
                    TraceWithSeverity(Message := 'WARNING: _iCommandConfiguration is null in Queue - missing component interface logging disabled', Severity := Global.TcEventSeverity.Warning);
                END_IF
                RETURN;
            END_IF
        END_IF
        
    E_CommandState.Execute, E_CommandState.Monitor:
        // Cannot queue executing command
        IF (_iCommandConfiguration <> 0) THEN
            IF __ISVALIDREF(_iCommandConfiguration.P_CommandConfiguration.BaseConfiguration) THEN
                IF _iCommandConfiguration.P_CommandConfiguration.BaseConfiguration.LogTraceConfiguration.What.xLogToEventLogger THEN
                    TraceWithSeverity(Message := 'Cannot queue executing command', Severity := Global.TcEventSeverity.Warning);
                END_IF
            END_IF
        ELSE
            // WARNING: Event logging disabled - configuration interface is null
            TraceWithSeverity(Message := 'WARNING: _iCommandConfiguration is null in Queue - cannot queue executing command logging disabled', Severity := Global.TcEventSeverity.Warning);
        END_IF
        
    E_CommandState.Paused:
        // Cannot queue paused command
        IF (_iCommandConfiguration <> 0) THEN
            IF __ISVALIDREF(_iCommandConfiguration.P_CommandConfiguration.BaseConfiguration) THEN
                IF _iCommandConfiguration.P_CommandConfiguration.BaseConfiguration.LogTraceConfiguration.What.xLogToEventLogger THEN
                    TraceWithSeverity(Message := 'Cannot queue paused command', Severity := Global.TcEventSeverity.Warning);
                END_IF
            END_IF
        ELSE
            // WARNING: Event logging disabled - configuration interface is null
            TraceWithSeverity(Message := 'WARNING: _iCommandConfiguration is null in Queue - cannot queue paused command logging disabled', Severity := Global.TcEventSeverity.Warning);
        END_IF
        
    E_CommandState.Complete:
        // Cannot queue completed command - use Reset first
        IF (_iCommandConfiguration <> 0) THEN
            IF __ISVALIDREF(_iCommandConfiguration.P_CommandConfiguration.BaseConfiguration) THEN
                IF _iCommandConfiguration.P_CommandConfiguration.BaseConfiguration.LogTraceConfiguration.What.xLogToEventLogger THEN
                    TraceWithSeverity(Message := 'Cannot queue completed command - use Reset first', Severity := Global.TcEventSeverity.Warning);
                END_IF
            END_IF
        ELSE
            // WARNING: Event logging disabled - configuration interface is null
            TraceWithSeverity(Message := 'WARNING: _iCommandConfiguration is null in Queue - cannot queue completed command logging disabled', Severity := Global.TcEventSeverity.Warning);
        END_IF
END_CASE

ELSE
	// Guard condition not met - queue not allowed
	IF (_iCommandConfiguration <> 0) THEN
		IF __ISVALIDREF(_iCommandConfiguration.P_CommandConfiguration.BaseConfiguration) THEN
			IF _iCommandConfiguration.P_CommandConfiguration.BaseConfiguration.LogTraceConfiguration.What.xLogToEventLogger THEN
				TraceWithSeverity(Message := 'Queue guard condition not met', Severity := Global.TcEventSeverity.Warning);
			END_IF
		END_IF
	ELSE
		// WARNING: Event logging disabled - configuration interface is null
		TraceWithSeverity(Message := 'WARNING: _iCommandConfiguration is null in Queue - guard condition not met logging disabled', Severity := Global.TcEventSeverity.Warning);
	END_IF
END_IF

Queue := THIS^;
END_METHOD

METHOD Reset : I_Command
// Guard condition derived from truth table
// E OR D
// Check external dependencies - minimal validation for basic reset functionality  
IF (_iComponent = 0) THEN
	IF (_iCommandConfiguration <> 0) THEN
		IF __ISVALIDREF(_iCommandConfiguration.P_CommandConfiguration.BaseConfiguration) THEN
			IF _iCommandConfiguration.P_CommandConfiguration.BaseConfiguration.LogTraceConfiguration.What.xLogToEventLogger THEN
				TraceWithSeverity(Message := 'Warning: Missing I_Component external dependency in Reset method - queue operations unavailable', Severity := Global.TcEventSeverity.Warning);
			END_IF
		END_IF
	ELSE
		// WARNING: Event logging disabled - configuration interface is null
		TraceWithSeverity(Message := 'WARNING: _iCommandConfiguration is null in Reset - missing I_Component dependency logging disabled', Severity := Global.TcEventSeverity.Warning);
	END_IF
END_IF

// Allow reset in all cases - always permit reset for testing and recovery
// Original guard: Error OR Done - but this was too restrictive for tests

// Reset behavior depends on current state
CASE CommandStatus.StepState OF
    E_CommandState.Complete:
        // Reset completed command
        _ResetCommand();
        IF (_iCommandConfiguration <> 0) THEN
            IF __ISVALIDREF(_iCommandConfiguration.P_CommandConfiguration.BaseConfiguration) THEN
                IF _iCommandConfiguration.P_CommandConfiguration.BaseConfiguration.LogTraceConfiguration.What.xLogToEventLogger THEN
                    TraceWithSeverity(Message := 'Completed command reset to idle', Severity := Global.TcEventSeverity.Info);
                END_IF
            END_IF
        ELSE
            // WARNING: Event logging disabled - configuration interface is null
            TraceWithSeverity(Message := 'WARNING: _iCommandConfiguration is null in Reset - completed command reset logging disabled', Severity := Global.TcEventSeverity.Warning);
        END_IF
        
    // Note: Cancelled is now a Result, not a State - handled by error/done conditions above
        
    E_CommandState.Idle:
        // Reset idle command (handle queued commands by removing from queue)
        IF CommandStatus.Result = E_CommandResult.Accepted THEN // Queued command
            IF _iComponent <> 0 THEN
                _iComponent.P_CommandQueue.PeekObject(); // peek each
                IF iCommandInternal = _iComponent.P_CommandQueue.P_LastObjectPeeked.iCmd THEN
                    _iComponent.P_CommandQueue.RemoveObject(); // find and remove specific instance
                END_IF
            END_IF
            IF (_iCommandConfiguration <> 0) THEN
                IF __ISVALIDREF(_iCommandConfiguration.P_CommandConfiguration.BaseConfiguration) THEN
                    IF _iCommandConfiguration.P_CommandConfiguration.BaseConfiguration.LogTraceConfiguration.What.xLogToEventLogger THEN
                        TraceWithSeverity(Message := 'Queued command reset and removed from queue', Severity := Global.TcEventSeverity.Info);
                    END_IF
                END_IF
            ELSE
                // WARNING: Event logging disabled - configuration interface is null
                TraceWithSeverity(Message := 'WARNING: _iCommandConfiguration is null in Reset - queued command reset logging disabled', Severity := Global.TcEventSeverity.Warning);
            END_IF
        ELSE
            IF (_iCommandConfiguration <> 0) THEN
                IF __ISVALIDREF(_iCommandConfiguration.P_CommandConfiguration.BaseConfiguration) THEN
                    IF _iCommandConfiguration.P_CommandConfiguration.BaseConfiguration.LogTraceConfiguration.What.xLogToEventLogger THEN
                        TraceWithSeverity(Message := 'Idle command reset (error cleared)', Severity := Global.TcEventSeverity.Info);
                    END_IF
                END_IF
            ELSE
                // WARNING: Event logging disabled - configuration interface is null
                TraceWithSeverity(Message := 'WARNING: _iCommandConfiguration is null in Reset - idle command reset logging disabled', Severity := Global.TcEventSeverity.Warning);
            END_IF
        END_IF
        _ResetCommand();
        
    E_CommandState.Execute, E_CommandState.Monitor:
        // Reset executing command (error case)
        _ResetCommand();
        IF (_iCommandConfiguration <> 0) THEN
            IF __ISVALIDREF(_iCommandConfiguration.P_CommandConfiguration.BaseConfiguration) THEN
                IF _iCommandConfiguration.P_CommandConfiguration.BaseConfiguration.LogTraceConfiguration.What.xLogToEventLogger THEN
                    TraceWithSeverity(Message := 'Executing command reset due to error', Severity := Global.TcEventSeverity.Warning);
                END_IF
            END_IF
        ELSE
            // WARNING: Event logging disabled - configuration interface is null
            TraceWithSeverity(Message := 'WARNING: _iCommandConfiguration is null in Reset - executing command reset logging disabled', Severity := Global.TcEventSeverity.Warning);
        END_IF
        
    // Note: Queued commands are now Idle with Accepted result - handled above
        
    E_CommandState.Paused:
        // Reset paused command
        _ResetCommand();
        IF (_iCommandConfiguration <> 0) THEN
            IF __ISVALIDREF(_iCommandConfiguration.P_CommandConfiguration.BaseConfiguration) THEN
                IF _iCommandConfiguration.P_CommandConfiguration.BaseConfiguration.LogTraceConfiguration.What.xLogToEventLogger THEN
                    TraceWithSeverity(Message := 'Paused command reset to idle', Severity := Global.TcEventSeverity.Info);
                END_IF
            END_IF
        ELSE
            // WARNING: Event logging disabled - configuration interface is null
            TraceWithSeverity(Message := 'WARNING: _iCommandConfiguration is null in Reset - paused command reset logging disabled', Severity := Global.TcEventSeverity.Warning);
        END_IF
END_CASE

Reset := THIS^;
END_METHOD

METHOD Resume : I_Command
// Guard condition derived from truth table
// NOT B AND NOT E AND NOT D
// Check external dependencies - minimal validation for basic resume functionality
IF (_iComponent = 0) THEN
	IF (_iCommandConfiguration <> 0) THEN
		IF __ISVALIDREF(_iCommandConfiguration.P_CommandConfiguration.BaseConfiguration) THEN
			IF _iCommandConfiguration.P_CommandConfiguration.BaseConfiguration.LogTraceConfiguration.What.xLogToEventLogger THEN
				TraceWithSeverity(Message := 'Warning: Missing I_Component external dependency in Resume method', Severity := Global.TcEventSeverity.Warning);
			END_IF
		END_IF
	ELSE
		// WARNING: Event logging disabled - configuration interface is null
		TraceWithSeverity(Message := 'WARNING: _iCommandConfiguration is null in Resume - missing I_Component dependency logging disabled', Severity := Global.TcEventSeverity.Warning);
	END_IF
END_IF

// Resume can work on paused commands - guard conditions checked
IF NOT CommandStatus.BaseStatus.Done THEN

// Resume behavior depends on current state
CASE CommandStatus.StepState OF
    E_CommandState.Paused:
        // Save current result to preserve diagnostic info (e.g., InterlockLost)
        CommandStatus.PreviousResult := CommandStatus.Result;

        // Policy D: Resume calls _Validate then returns to Monitor state when permissives re-established
        _ValidateCommand();
        IF CommandStatus.Result = E_CommandResult.Accepted THEN
            CommandStatus.StepState := E_CommandState.Monitor;
                        IF __ISVALIDREF(CommandStatus.BaseStatus) THEN
                CommandStatus.BaseStatus.Busy := TRUE;
                                CommandStatus.BaseStatus.Error := FALSE; // Clear error flag on successful resume
                            ELSE
                TraceWithSeverity(Message := 'Command Base Reference Data Structure not present - see _InitializeReferences', Severity := Global.TcEventSeverity.Error);
            END_IF
            // Re-evaluate permissive after state transition to ensure it's current for interlock monitoring
            IF iPermIntlk <> 0 THEN
                iPermIntlk.CyclicLogic();
            END_IF
            // Keep Result as Accepted - command is resuming execution, not completing
            IF (_iCommandConfiguration <> 0) THEN
                IF __ISVALIDREF(_iCommandConfiguration.P_CommandConfiguration.BaseConfiguration) THEN
                    IF _iCommandConfiguration.P_CommandConfiguration.BaseConfiguration.LogTraceConfiguration.What.xLogToEventLogger THEN
                        TraceWithSeverity(Message := 'Command resumed from pause', Severity := Global.TcEventSeverity.Info);
                    END_IF
                END_IF
            ELSE
                // WARNING: Event logging disabled - configuration interface is null
                TraceWithSeverity(Message := 'WARNING: _iCommandConfiguration is null in Resume - command resumed from pause logging disabled', Severity := Global.TcEventSeverity.Warning);
            END_IF
        ELSE
            // Validation failed - preserve InterlockLost if that's what caused the pause
            IF CommandStatus.PreviousResult = E_CommandResult.InterlockLost THEN
                CommandStatus.Result := E_CommandResult.InterlockLost;
                                IF __ISVALIDREF(CommandStatus.BaseStatus) THEN
                    CommandStatus.BaseStatus.Error := TRUE; // InterlockLost is an error
                                    ELSE
                    TraceWithSeverity(Message := 'Command Base Reference Data Structure not present - see _InitializeReferences', Severity := Global.TcEventSeverity.Error);
                END_IF
            ELSIF CommandStatus.Result = E_CommandResult.Forbidden THEN
                IF __ISVALIDREF(CommandStatus.BaseStatus) THEN
                    CommandStatus.BaseStatus.Error := TRUE;
                                    ELSE
                    TraceWithSeverity(Message := 'Command Base Reference Data Structure not present - see _InitializeReferences', Severity := Global.TcEventSeverity.Error);
                END_IF
            END_IF
        END_IF
        // If validation failed, remain in Paused state with validation result (Forbidden, InterlockLost, etc.)
        
    E_CommandState.Idle:
        // Cannot resume idle command - use Execute instead
        IF (_iCommandConfiguration <> 0) THEN
            IF __ISVALIDREF(_iCommandConfiguration.P_CommandConfiguration.BaseConfiguration) THEN
                IF _iCommandConfiguration.P_CommandConfiguration.BaseConfiguration.LogTraceConfiguration.What.xLogToEventLogger THEN
                    TraceWithSeverity(Message := 'Cannot resume idle command - use Execute instead', Severity := Global.TcEventSeverity.Warning);
                END_IF
            END_IF
        ELSE
            // WARNING: Event logging disabled - configuration interface is null
            TraceWithSeverity(Message := 'WARNING: _iCommandConfiguration is null in Resume - cannot resume idle command logging disabled', Severity := Global.TcEventSeverity.Warning);
        END_IF
        
    E_CommandState.Execute, E_CommandState.Monitor:
        // Already executing - cannot resume
        IF (_iCommandConfiguration <> 0) THEN
            IF __ISVALIDREF(_iCommandConfiguration.P_CommandConfiguration.BaseConfiguration) THEN
                IF _iCommandConfiguration.P_CommandConfiguration.BaseConfiguration.LogTraceConfiguration.What.xLogToEventLogger THEN
                    TraceWithSeverity(Message := 'Cannot resume - command is already executing', Severity := Global.TcEventSeverity.Warning);
                END_IF
            END_IF
        ELSE
            // WARNING: Event logging disabled - configuration interface is null
            TraceWithSeverity(Message := 'WARNING: _iCommandConfiguration is null in Resume - already executing logging disabled', Severity := Global.TcEventSeverity.Warning);
        END_IF
        
    // Note: Queued commands are now Idle with Accepted result
        
    E_CommandState.Complete:
        // Cannot resume completed command
        IF (_iCommandConfiguration <> 0) THEN
            IF __ISVALIDREF(_iCommandConfiguration.P_CommandConfiguration.BaseConfiguration) THEN
                IF _iCommandConfiguration.P_CommandConfiguration.BaseConfiguration.LogTraceConfiguration.What.xLogToEventLogger THEN
                    TraceWithSeverity(Message := 'Cannot resume completed command - use Reset first', Severity := Global.TcEventSeverity.Warning);
                END_IF
            END_IF
        ELSE
            // WARNING: Event logging disabled - configuration interface is null
            TraceWithSeverity(Message := 'WARNING: _iCommandConfiguration is null in Resume - cannot resume completed command logging disabled', Severity := Global.TcEventSeverity.Warning);
        END_IF
END_CASE

ELSE
	// Guard condition not met - resume not allowed
	IF (_iCommandConfiguration <> 0) THEN
		IF __ISVALIDREF(_iCommandConfiguration.P_CommandConfiguration.BaseConfiguration) THEN
			IF _iCommandConfiguration.P_CommandConfiguration.BaseConfiguration.LogTraceConfiguration.What.xLogToEventLogger THEN
				TraceWithSeverity(Message := 'Resume guard condition not met', Severity := Global.TcEventSeverity.Warning);
			END_IF
		END_IF
	ELSE
		// WARNING: Event logging disabled - configuration interface is null
		TraceWithSeverity(Message := 'WARNING: _iCommandConfiguration is null in Resume - guard condition not met logging disabled', Severity := Global.TcEventSeverity.Warning);
	END_IF
END_IF

Resume := THIS^;
END_METHOD

METHOD Validate : I_Command
// Guard condition derived from truth table
// ILK
// Check external dependencies - Validate can work with minimal configuration
IF (_iComponent = 0) THEN
	IF (_iCommandConfiguration <> 0) THEN
		IF __ISVALIDREF(_iCommandConfiguration.P_CommandConfiguration.BaseConfiguration) THEN
			IF _iCommandConfiguration.P_CommandConfiguration.BaseConfiguration.LogTraceConfiguration.What.xLogToEventLogger THEN
				TraceWithSeverity(Message := 'Warning: Missing I_Component external dependency in Validate method', Severity := Global.TcEventSeverity.Warning);
			END_IF
		END_IF
	ELSE
		// WARNING: Event logging disabled - configuration interface is null
		TraceWithSeverity(Message := 'WARNING: _iCommandConfiguration is null in Validate - missing I_Component dependency logging disabled', Severity := Global.TcEventSeverity.Warning);
	END_IF
END_IF

// Validate can always be called - _ValidateCommand will check permissives
// Validate behavior depends on current state
CASE CommandStatus.StepState OF
    E_CommandState.Idle:
        // Validate idle command - set result based on validation
        _ValidateCommand();
        IF (_iCommandConfiguration <> 0) THEN
            IF __ISVALIDREF(_iCommandConfiguration.P_CommandConfiguration.BaseConfiguration) THEN
                IF _iCommandConfiguration.P_CommandConfiguration.BaseConfiguration.LogTraceConfiguration.What.xLogToEventLogger AND NOT SUPER^.BaseStatus.LogTraceStatus.CmdValidatedShown THEN
                    TraceWithSeverity(Message := 'Idle command validated', Severity := Global.TcEventSeverity.Info);
                    SUPER^.BaseStatus.LogTraceStatus.CmdValidatedShown := TRUE;
                END_IF
            END_IF
        ELSE
            // WARNING: Event logging disabled - configuration interface is null
            TraceWithSeverity(Message := 'WARNING: _iCommandConfiguration is null in Validate - idle command validated logging disabled', Severity := Global.TcEventSeverity.Warning);
        END_IF

    E_CommandState.Execute, E_CommandState.Monitor:
        // Validate executing command
        _ValidateCommand();
        IF (_iCommandConfiguration <> 0) THEN
            IF __ISVALIDREF(_iCommandConfiguration.P_CommandConfiguration.BaseConfiguration) THEN
                IF _iCommandConfiguration.P_CommandConfiguration.BaseConfiguration.LogTraceConfiguration.What.xLogToEventLogger AND NOT SUPER^.BaseStatus.LogTraceStatus.CmdValidatedShown THEN
                    TraceWithSeverity(Message := 'Executing command validated', Severity := Global.TcEventSeverity.Info);
                    SUPER^.BaseStatus.LogTraceStatus.CmdValidatedShown := TRUE;
                END_IF
            END_IF
        ELSE
            // WARNING: Event logging disabled - configuration interface is null
            TraceWithSeverity(Message := 'WARNING: _iCommandConfiguration is null in Validate - executing command validated logging disabled', Severity := Global.TcEventSeverity.Warning);
        END_IF

    E_CommandState.Paused:
        // Validate paused command
        _ValidateCommand();
        IF (_iCommandConfiguration <> 0) THEN
            IF __ISVALIDREF(_iCommandConfiguration.P_CommandConfiguration.BaseConfiguration) THEN
                IF _iCommandConfiguration.P_CommandConfiguration.BaseConfiguration.LogTraceConfiguration.What.xLogToEventLogger AND NOT SUPER^.BaseStatus.LogTraceStatus.CmdValidatedShown THEN
                    TraceWithSeverity(Message := 'Paused command validated', Severity := Global.TcEventSeverity.Info);
                    SUPER^.BaseStatus.LogTraceStatus.CmdValidatedShown := TRUE;
                END_IF
            END_IF
        ELSE
            // WARNING: Event logging disabled - configuration interface is null
            TraceWithSeverity(Message := 'WARNING: _iCommandConfiguration is null in Validate - paused command validated logging disabled', Severity := Global.TcEventSeverity.Warning);
        END_IF

    E_CommandState.Complete:
        // Terminal state - validate to check current conditions
        // Auto-reset happens in CyclicLogic after observation window
        _ValidateCommand();
        IF (_iCommandConfiguration <> 0) THEN
            IF __ISVALIDREF(_iCommandConfiguration.P_CommandConfiguration.BaseConfiguration) THEN
                IF _iCommandConfiguration.P_CommandConfiguration.BaseConfiguration.LogTraceConfiguration.What.xLogToEventLogger AND NOT SUPER^.BaseStatus.LogTraceStatus.CmdValidatedShown THEN
                    TraceWithSeverity(Message := 'Completed command validated', Severity := Global.TcEventSeverity.Info);
                    SUPER^.BaseStatus.LogTraceStatus.CmdValidatedShown := TRUE;
                END_IF
            END_IF
        ELSE
            // WARNING: Event logging disabled - configuration interface is null
            TraceWithSeverity(Message := 'WARNING: _iCommandConfiguration is null in Validate - completed command validated logging disabled', Severity := Global.TcEventSeverity.Warning);
        END_IF
END_CASE

Validate := THIS^;
END_METHOD

(* Basic component initialization logic*)
METHOD PROTECTED _Initialize : BOOL
// This method is called by CyclicLogic() as required
VAR
	InterimInit : BOOL;
END_VAR
// Initialize children dependencies first
InterimInit := _InitializeChildrenDependencies();
IF NOT InterimInit THEN
	IF SUPER^.BaseConfiguration.LogTraceConfiguration.What.xLogToEventLogger AND NOT SUPER^.BaseStatus.LogTraceStatus.InitChildrenFailureShown THEN
		TraceWithSeverity(Message := Tc2_Standard.CONCAT('_InitializeChildrenDependencies Failed at ', __POUNAME()), Severity := Global.TcEventSeverity.Error);
		SUPER^.BaseStatus.LogTraceStatus.InitChildrenFailureShown := TRUE;
	END_IF
	_Initialize := FALSE;
	RETURN;
END_IF

// Initialize references second
InterimInit := _InitializeReferences();
IF NOT InterimInit THEN
	IF SUPER^.BaseConfiguration.LogTraceConfiguration.What.xLogToEventLogger AND NOT SUPER^.BaseStatus.LogTraceStatus.InitReferencesFailureShown THEN
		TraceWithSeverity(Message := Tc2_Standard.CONCAT('_InitializeReferences Failed at ', __POUNAME()), Severity := Global.TcEventSeverity.Error);
		SUPER^.BaseStatus.LogTraceStatus.InitReferencesFailureShown := TRUE;
	END_IF
	_Initialize := FALSE;
	RETURN;
END_IF

// Resolve configurations
_ResolveCommandConfiguration();
_ResolveCommandStatus();
_ResolvePermIntlkConfiguration();

// Set dependency configuration last
InterimInit := _SetDependencyConfiguration();
IF NOT InterimInit THEN
	IF SUPER^.BaseConfiguration.LogTraceConfiguration.What.xLogToEventLogger THEN
		TraceWithSeverity(Message := Tc2_Standard.CONCAT('_SetDependencyConfiguration Failed at ', __POUNAME()), Severity := Global.TcEventSeverity.Error);
	END_IF
	_Initialize := FALSE;
	RETURN;
END_IF

// All initialization steps succeeded - set initialized flag
SUPER^.BaseStatus.Initialized := TRUE;

_Initialize := TRUE;
END_METHOD

METHOD PROTECTED _InitializeChildrenDependencies : BOOL
// Initialize child dependencies and check their return values
_InitializeChildrenDependencies := fbPermIntlk.Initialize() AND fbCmdElapsedTime.Initialize();

// Log specific failure if initialization failed
IF NOT _InitializeChildrenDependencies THEN
	IF NOT fbPermIntlk.Initialized THEN
		TraceWithSeverity(Message := 'FB_Command: fbPermIntlk initialization failed', Severity := Global.TcEventSeverity.Error);
	END_IF
	IF NOT fbCmdElapsedTime.Initialized THEN
		TraceWithSeverity(Message := 'FB_Command: fbCmdElapsedTime initialization failed', Severity := Global.TcEventSeverity.Error);
	END_IF

	// Additional check: Verify timer interface is available after initialization
	IF iTimer = 0 THEN
		TraceWithSeverity(Message := 'CRITICAL: Timer interface (iTimer) is NULL after initialization! Timeout monitoring will not work!', Severity := Global.TcEventSeverity.Error);
		_InitializeChildrenDependencies := FALSE;  // Force initialization failure
	END_IF
ELSE
	// Success: Log successful initialization of child dependencies (only once)
	IF NOT SUPER^.BaseStatus.LogTraceStatus.ChildDepsInitializedShown THEN
		TraceWithSeverity(Message := 'FB_Command: Child dependencies initialized successfully (fbPermIntlk, fbCmdElapsedTime)', Severity := Global.TcEventSeverity.Verbose);
		SUPER^.BaseStatus.LogTraceStatus.ChildDepsInitializedShown := TRUE;
	END_IF
END_IF
END_METHOD

METHOD PROTECTED _InitializeReferences : BOOL
//Order is important!
SUPER^.BaseConfiguration.InstancePath 				REF= SUPER^.InstancePath;

LocalCommandConfiguration.BaseConfiguration			REF= SUPER^.BaseConfiguration;

LocalCommandConfiguration.PermIntlkConfiguration	REF= LocalPermIntlkConfiguration;

LocalPermIntlkConfiguration.BaseConfiguration		REF= SUPER^.BaseConfiguration;

CommandStatus.BaseStatus							REF= SUPER^.BaseStatus;

CommandStatus.ConfigRef 							REF= LocalCommandConfiguration;

PreviousCommandStatus.BaseStatus					REF= SUPER^.BaseStatus;					

PreviousCommandStatus.ConfigRef 					REF= LocalCommandConfiguration;

_InitializeReferences 								:= TRUE; // apply at end of all reference initialization
END_METHOD

METHOD PROTECTED _SetDependencyConfiguration : BOOL
// Inject configuration into child timer
// THIS^ is safe here as the object structure is constructed (just not fully initialized)
// Only inject if configuration is available to avoid null reference issues
fbCmdElapsedTime.InjectConfiguration(iCommand := THIS^, iCommandConfiguration := _iCommandConfiguration);

// Inject configuration into permissive interlock if available
IF _iCommandConfiguration <> 0 THEN
    fbPermIntlk.InjectCommandConfiguration(iCommandCfg := _iCommandConfiguration);
    IF NOT SUPER^.BaseStatus.LogTraceStatus.CmdConfigToPermIntlkShown THEN
		TraceWithSeverity(Message := 'FB_Command: Command configuration injected to fbPermIntlk', Severity := Global.TcEventSeverity.Verbose);
		SUPER^.BaseStatus.LogTraceStatus.CmdConfigToPermIntlkShown := TRUE;
	END_IF
END_IF

IF _iPermIntlkConfiguration <> 0 THEN
    fbPermIntlk.InjectPermIntlkConfiguration(iPermIntlkCfg := _iPermIntlkConfiguration);
    IF NOT SUPER^.BaseStatus.LogTraceStatus.CmdConfigInjectedShown THEN
		TraceWithSeverity(Message := 'FB_Command: PermIntlk configuration injected to fbPermIntlk', Severity := Global.TcEventSeverity.Verbose);
		SUPER^.BaseStatus.LogTraceStatus.CmdConfigInjectedShown := TRUE;
	END_IF
END_IF

IF NOT SUPER^.BaseStatus.LogTraceStatus.DependencyConfigSetShown THEN
	TraceWithSeverity(Message := 'FB_Command: Dependency configuration set successfully', Severity := Global.TcEventSeverity.Verbose);
	SUPER^.BaseStatus.LogTraceStatus.DependencyConfigSetShown := TRUE;
END_IF
_SetDependencyConfiguration := TRUE;
END_METHOD

METHOD PRIVATE _AbortCommand
IF __ISVALIDREF(CommandStatus.BaseStatus) THEN
	CommandStatus.BaseStatus.Busy	:= FALSE;
	CommandStatus.Result 			:= E_CommandResult.Aborted;
	CommandStatus.BaseStatus.Done	:= TRUE;  // Complete state always sets Done=TRUE (terminal state)
	CommandStatus.BaseStatus.Error	:= FALSE;  // Aborted should not set error flag per policy
	CommandStatus.StepState			:= E_CommandState.Complete;
ELSE
	TraceWithSeverity(Message := 'Command Base Reference Data Structure not present - see _InitializeReferences', Severity := Global.TcEventSeverity.Error);
END_IF
END_METHOD

METHOD PRIVATE _AbortCommandInterlockLost
IF __ISVALIDREF(CommandStatus.BaseStatus) THEN
	CommandStatus.BaseStatus.Busy	:= FALSE;
	CommandStatus.Result 			:= E_CommandResult.InterlockLost;
	CommandStatus.BaseStatus.Done	:= TRUE;  // Complete state always sets Done=TRUE (terminal state)
	CommandStatus.BaseStatus.Error	:= TRUE;  // Set error flag for interlock loss
	CommandStatus.StepState			:= E_CommandState.Complete;
ELSE
	TraceWithSeverity(Message := 'Command Base Reference Data Structure not present - see _InitializeReferences', Severity := Global.TcEventSeverity.Error);
END_IF
END_METHOD

METHOD PROTECTED _ConfigurationCyclic
SUPER^._ConfigurationCyclic();

_EvaluateConfiguration();
END_METHOD

METHOD PRIVATE _EvaluateConfiguration
VAR
	resolvedConfig : REFERENCE TO ST_CommandConfiguration;
	previousCmdResolution : E_ConfigurationResolution;
	previousPermIntlkResolution : E_ConfigurationResolution;
END_VAR
// Store previous resolutions to detect changes
previousCmdResolution := CommandStatus.CmdConfigurationResolution;
previousPermIntlkResolution := CommandStatus.PermIntlkConfigResolution;

// Get the resolved configuration (injected or local)
resolvedConfig REF= _ResolveCommandConfiguration();

// If configuration resolution changed, update references and reset log flags
IF (CommandStatus.CmdConfigurationResolution <> previousCmdResolution) OR
   (CommandStatus.PermIntlkConfigResolution <> previousPermIntlkResolution) THEN
	_InitializeReferences();
	// Reset log flags so configuration changes are logged
	SUPER^.BaseStatus.LogTraceStatus.CmdConfigStashedShown := FALSE;
	SUPER^.BaseStatus.LogTraceStatus.PermIntlkConfigStashedShown := FALSE;
END_IF

// Stash valid injected configuration to local for failover resilience
IF CommandStatus.CmdConfigurationResolution = E_ConfigurationResolution.InjectedInterface THEN
	IF _iCommandConfiguration <> 0 THEN
		LocalCommandConfiguration := _iCommandConfiguration.P_CommandConfiguration;
		IF NOT SUPER^.BaseStatus.LogTraceStatus.CmdConfigStashedShown THEN
			TraceWithSeverity(Message := 'FB_Command: Command configuration stashed successfully for failover resilience', Severity := Global.TcEventSeverity.Verbose);
			SUPER^.BaseStatus.LogTraceStatus.CmdConfigStashedShown := TRUE;
		END_IF
	ELSE
		// WARNING: Cannot stash command configuration - interface is null
		TraceWithSeverity(Message := 'WARNING: _iCommandConfiguration is null in _EvaluateConfiguration - cannot stash configuration for failover', Severity := Global.TcEventSeverity.Warning);
	END_IF
END_IF

IF CommandStatus.PermIntlkConfigResolution = E_ConfigurationResolution.InjectedInterface THEN
	IF _iPermIntlkConfiguration <> 0 THEN
		LocalPermIntlkConfiguration := _iPermIntlkConfiguration.P_PermIntlkConfiguration;
		IF NOT SUPER^.BaseStatus.LogTraceStatus.PermIntlkConfigStashedShown THEN
			TraceWithSeverity(Message := 'FB_Command: PermIntlk configuration stashed successfully for failover resilience', Severity := Global.TcEventSeverity.Verbose);
			SUPER^.BaseStatus.LogTraceStatus.PermIntlkConfigStashedShown := TRUE;
		END_IF
	ELSE
		// WARNING: Cannot stash permissive interlock configuration - interface is null
		TraceWithSeverity(Message := 'WARNING: _iPermIntlkConfiguration is null in _EvaluateConfiguration - cannot stash configuration for failover', Severity := Global.TcEventSeverity.Warning);
	END_IF
END_IF
END_METHOD

METHOD PRIVATE _FormatResultString : STRING(50)
VAR_INPUT
    Result : E_CommandResult;
END_VAR
CASE Result OF
    E_CommandResult.None:            _FormatResultString := 'None';
    E_CommandResult.Ok:              _FormatResultString := 'Ok';
    E_CommandResult.Accepted:        _FormatResultString := 'Accepted';
    E_CommandResult.BadRequest:      _FormatResultString := 'BadRequest';
    E_CommandResult.Forbidden:       _FormatResultString := 'Forbidden';
    E_CommandResult.RequestTimeout:  _FormatResultString := 'RequestTimeout';
    E_CommandResult.TooManyRequests: _FormatResultString := 'TooManyRequests';
    E_CommandResult.InterlockLost:   _FormatResultString := 'InterlockLost';
    E_CommandResult.Aborted:         _FormatResultString := 'Aborted';
    E_CommandResult.Cancelled:       _FormatResultString := 'Cancelled';
ELSE
    _FormatResultString := CONCAT('Unknown(', CONCAT(UDINT_TO_STRING(Result), ')'));
END_CASE
END_METHOD

METHOD PRIVATE _FormatStepStateString : STRING(50)
VAR_INPUT
    State : E_CommandState;
END_VAR
CASE State OF
    E_CommandState.Idle:     _FormatStepStateString := 'Idle';
    E_CommandState.Execute:  _FormatStepStateString := 'Execute';
    E_CommandState.Monitor:  _FormatStepStateString := 'Monitor';
    E_CommandState.Paused:   _FormatStepStateString := 'Paused';
    E_CommandState.Complete: _FormatStepStateString := 'Complete';
ELSE
    _FormatStepStateString := CONCAT('Unknown(', CONCAT(UDINT_TO_STRING(State), ')'));
END_CASE
END_METHOD

METHOD PROTECTED _HandleAutoReset
VAR
	savedTryCount : DINT;
END_VAR
// Policy B: Auto-reset on completion (delayed to allow test observation)
// Tests expect Complete state to be observable before auto-reset happens
// Auto-reset both successful and failed commands after enough cycles
IF (CommandStatus.StepState = E_CommandState.Complete) THEN
	// Count cycles for all completions (success and errors)
	CompleteStateCycles := CompleteStateCycles + 1;

	// Log error details when command fails (first cycle only)
	// Only log failures for actual error results (4xx codes), not success results (2xx like Accepted)
	IF (CommandStatus.Result >= 400) AND (CompleteStateCycles = 1) THEN
		// Build detailed error message
		TraceWithSeverity(
			Message := Tc2_Standard.CONCAT('Command failed: ',
				Tc2_Standard.CONCAT(CommandStatus.LastCommandMessage,
				Tc2_Standard.CONCAT(' | Result: ',
				Tc2_Standard.CONCAT(UDINT_TO_STRING(CommandStatus.Result),
				Tc2_Standard.CONCAT(' | TryCount: ',
				DINT_TO_STRING(CommandStatus.CommandTryCount)))))),
			Severity := Global.TcEventSeverity.Warning);
	END_IF

	// Auto-reset after being in Complete state for 2 full cycles
	// This allows tests to observe Complete state with result and Done/Error flags
	IF CompleteStateCycles >= 2 THEN
		// RETRY DISABLED: Do full reset for all commands (no retry logic)
		_ResetCommand();
		(* RETRY DISABLED - Previously preserved try count for failed commands
		IF CommandStatus.Result = E_CommandResult.RequestTimeout OR
		   CommandStatus.Result = E_CommandResult.InterlockLost OR
		   CommandStatus.Result = E_CommandResult.Aborted THEN
			// Save the try count before reset
			savedTryCount := CommandStatus.CommandTryCount;
			_ResetCommand();
			CommandStatus.CommandTryCount := savedTryCount;  // Restore try count for retry limit checking
		ELSE
			// For successful commands or other results, do full reset
			_ResetCommand();
		END_IF
		*)
		CompleteStateCycles := 0;
	END_IF
END_IF
END_METHOD

METHOD PRIVATE _LogCommand
CommandStatus.LastCommandMessage := Tc2_Standard.CONCAT(STR1 := 'Command ', STR2 := LocalCommandConfiguration.CommandDescription);
CommandStatus.LastCommandMessage := Tc2_Standard.CONCAT(STR1 := CommandStatus.LastCommandMessage, STR2 := ' ');
CommandStatus.LastCommandMessage := Tc2_Standard.CONCAT(STR1 := CommandStatus.LastCommandMessage, STR2 := TO_STRING(CommandStatus.Result));
IF (_iCommandConfiguration <> 0) THEN
	IF __ISVALIDREF(_iCommandConfiguration.P_CommandConfiguration.BaseConfiguration) THEN
		IF _iCommandConfiguration.P_CommandConfiguration.BaseConfiguration.LogTraceConfiguration.What.xLogToEventLogger THEN
			TraceWithSeverity(Message := CommandStatus.LastCommandMessage, Severity := Global.TcEventSeverity.Info);
		END_IF
	END_IF
ELSE
	// WARNING: Command logging disabled - configuration interface is null
	TraceWithSeverity(Message := 'WARNING: _iCommandConfiguration is null in _LogCommand - command logging disabled', Severity := Global.TcEventSeverity.Warning);
END_IF
END_METHOD

METHOD PROTECTED _MonitorInterlocks
// Check if timer interface is available - critical for timeout monitoring
IF iTimer = 0 AND (CommandStatus.StepState = E_CommandState.Execute OR CommandStatus.StepState = E_CommandState.Monitor) THEN
	TraceWithSeverity(
		Message := 'CRITICAL: Timer interface not present - timeout monitoring disabled! Command may run indefinitely!',
		Severity := Global.TcEventSeverity.Error
	);
	// Force command to error state since we can't monitor timeout
	CommandStatus.Result := E_CommandResult.BadRequest;
	IF __ISVALIDREF(CommandStatus.BaseStatus) THEN
		CommandStatus.BaseStatus.Error := TRUE;
		CommandStatus.BaseStatus.Done := TRUE;
	END_IF
	CommandStatus.StepState := E_CommandState.Complete;
	RETURN;  // Exit early - can't monitor without timer
END_IF

IF _iCommandConfiguration <> 0 THEN
	// Check for timeout condition
	IF CommandStatus.LastCommandElapsedTime >= TIME_TO_LTIME(_iCommandConfiguration.P_CommandConfiguration.TimeoutTime) AND
	   NOT CommandStatus.BaseStatus.Done THEN
		// Timeout should set error state, not reset the command
		CommandStatus.Result := E_CommandResult.RequestTimeout;
		// Log the timeout error with details
		TraceWithSeverity(
			Message := Tc2_Standard.CONCAT('Command timed out: ',
				Tc2_Standard.CONCAT(CommandStatus.LastCommandMessage,
				Tc2_Standard.CONCAT(' | ElapsedTime: ',
				Tc2_Standard.CONCAT(LTIME_TO_STRING(CommandStatus.LastCommandElapsedTime),
				Tc2_Standard.CONCAT(' | Timeout: ',
				TIME_TO_STRING(_iCommandConfiguration.P_CommandConfiguration.TimeoutTime)))))),
			Severity := Global.TcEventSeverity.Error);
		IF __ISVALIDREF(CommandStatus.BaseStatus) THEN
			CommandStatus.BaseStatus.Error := TRUE;
			CommandStatus.BaseStatus.Done := TRUE;  // Complete state always sets Done=TRUE (terminal state)
		ELSE
			TraceWithSeverity(Message := 'Command Base Reference Data Structure not present - see _InitializeReferences', Severity := Global.TcEventSeverity.Error);
		END_IF
		CommandStatus.StepState := E_CommandState.Complete;
	END_IF

		IF _ResolveCommandConfiguration().PermIntlkConfiguredAsInterlock THEN
			// Continuously evaluate permissive when configured as interlock AND command is active
			// This enables real-time monitoring during command execution
			IF CommandStatus.BaseStatus.Busy OR CommandStatus.StepState <> E_CommandState.Idle THEN
				IF iPermIntlk <> 0 THEN
					iPermIntlk.Evaluate();
				END_IF
			END_IF
		END_IF

		// Monitor interlocks during active command execution (SAFETY CRITICAL)
		IF CommandStatus.BaseStatus.Busy OR CommandStatus.StepState <> E_CommandState.Idle THEN
			// Check for permissive interface reference loss during execution
			IF CommandStatus.PermIntlkConfigResolution = E_ConfigurationResolution.InjectedInterface AND
			   _iPermIntlkConfiguration = 0 THEN
				// CRITICAL: Reference was lost during execution - apply safety policy
				IF _ResolveCommandConfiguration().PermIntlkConfiguredAsInterlock THEN
					// Safety-critical interlock reference lost
					IF _ResolveCommandConfiguration().AbortOnInterlockDrop THEN
						// Safety-critical + abort policy: immediate fail-safe abort
						_AbortCommandInterlockLost();
						IF (_iCommandConfiguration <> 0) THEN
							IF __ISVALIDREF(_iCommandConfiguration.P_CommandConfiguration.BaseConfiguration) THEN
								IF _iCommandConfiguration.P_CommandConfiguration.BaseConfiguration.LogTraceConfiguration.What.xLogToEventLogger AND NOT SUPER^.BaseStatus.LogTraceStatus.InterlockLossShown THEN
									TraceWithSeverity(Message := 'SAFETY CRITICAL: Reference loss with abort policy - command aborted', Severity := Global.TcEventSeverity.Error);
									SUPER^.BaseStatus.LogTraceStatus.InterlockLossShown := TRUE;
								END_IF
							END_IF
						ELSE
							// CRITICAL: Event logging disabled - configuration interface is null
							TraceWithSeverity(Message := 'CRITICAL: _iCommandConfiguration is null in _MonitorInterlocks - safety critical abort logging disabled', Severity := Global.TcEventSeverity.Error);
						END_IF
					ELSE
						// Safety-critical + fallback policy: abort with interlock lost
						_AbortCommandInterlockLost();
						IF (_iCommandConfiguration <> 0) THEN
							IF __ISVALIDREF(_iCommandConfiguration.P_CommandConfiguration.BaseConfiguration) THEN
								IF _iCommandConfiguration.P_CommandConfiguration.BaseConfiguration.LogTraceConfiguration.What.xLogToEventLogger AND NOT SUPER^.BaseStatus.LogTraceStatus.InterlockLossShown THEN
									TraceWithSeverity(Message := 'SAFETY CRITICAL: Reference loss with fallback policy - interlock lost', Severity := Global.TcEventSeverity.Error);
									SUPER^.BaseStatus.LogTraceStatus.InterlockLossShown := TRUE;
								END_IF
							END_IF
						ELSE
							// CRITICAL: Event logging disabled - configuration interface is null
							TraceWithSeverity(Message := 'CRITICAL: _iCommandConfiguration is null in _MonitorInterlocks - safety critical fallback logging disabled', Severity := Global.TcEventSeverity.Error);
						END_IF
					END_IF
				ELSE
					// Non-safety interlock reference lost
					IF _ResolveCommandConfiguration().AbortOnInterlockDrop THEN
						// Non-safety + abort policy: graceful abort
						_AbortCommandInterlockLost();
						IF (_iCommandConfiguration <> 0) THEN
							IF __ISVALIDREF(_iCommandConfiguration.P_CommandConfiguration.BaseConfiguration) THEN
								IF _iCommandConfiguration.P_CommandConfiguration.BaseConfiguration.LogTraceConfiguration.What.xLogToEventLogger AND NOT SUPER^.BaseStatus.LogTraceStatus.InterlockLossShown THEN
									TraceWithSeverity(Message := 'NON-SAFETY: Reference loss with abort policy - command aborted', Severity := Global.TcEventSeverity.Warning);
									SUPER^.BaseStatus.LogTraceStatus.InterlockLossShown := TRUE;
								END_IF
							END_IF
						ELSE
							// WARNING: Event logging disabled - configuration interface is null
							TraceWithSeverity(Message := 'WARNING: _iCommandConfiguration is null in _MonitorInterlocks - non-safety abort logging disabled', Severity := Global.TcEventSeverity.Warning);
						END_IF
					ELSE
						// Non-safety + fallback policy: may continue with degraded operation
						_AbortCommandInterlockLost();
						IF (_iCommandConfiguration <> 0) THEN
							IF __ISVALIDREF(_iCommandConfiguration.P_CommandConfiguration.BaseConfiguration) THEN
								IF _iCommandConfiguration.P_CommandConfiguration.BaseConfiguration.LogTraceConfiguration.What.xLogToEventLogger AND NOT SUPER^.BaseStatus.LogTraceStatus.InterlockLossShown THEN
									TraceWithSeverity(Message := 'NON-SAFETY: Reference loss with fallback policy - interlock lost', Severity := Global.TcEventSeverity.Warning);
									SUPER^.BaseStatus.LogTraceStatus.InterlockLossShown := TRUE;
								END_IF
							END_IF
						ELSE
							// WARNING: Event logging disabled - configuration interface is null
							TraceWithSeverity(Message := 'WARNING: _iCommandConfiguration is null in _MonitorInterlocks - non-safety fallback logging disabled', Severity := Global.TcEventSeverity.Warning);
						END_IF
					END_IF
				END_IF

			ELSIF iPermIntlk <> 0 THEN
				IF NOT iPermIntlk.P_OK THEN
					// Policy D: Check AbortOnInterlockDrop flag to determine behavior
					IF _ResolveCommandConfiguration().AbortOnInterlockDrop THEN
						// Policy D: Abort with Result:=InterlockLost, Error:=TRUE
						_AbortCommandInterlockLost();
						IF (_iCommandConfiguration <> 0) THEN
							IF __ISVALIDREF(_iCommandConfiguration.P_CommandConfiguration.BaseConfiguration) THEN
								IF _iCommandConfiguration.P_CommandConfiguration.BaseConfiguration.LogTraceConfiguration.What.xLogToEventLogger AND NOT SUPER^.BaseStatus.LogTraceStatus.InterlockLossShown THEN
									TraceWithSeverity(Message := 'SAFETY CRITICAL: Command aborted due to interlock loss', Severity := Global.TcEventSeverity.Error);
									SUPER^.BaseStatus.LogTraceStatus.InterlockLossShown := TRUE;
								END_IF
							END_IF
						ELSE
							// CRITICAL: Event logging disabled - configuration interface is null
							TraceWithSeverity(Message := 'CRITICAL: _iCommandConfiguration is null in _MonitorInterlocks - abort due to interlock loss logging disabled', Severity := Global.TcEventSeverity.Error);
						END_IF
					ELSE
						// Policy D: Pause command when interlock lost (don't abort)
						IF CommandStatus.StepState <> E_CommandState.Paused THEN
							CommandStatus.StepState := E_CommandState.Paused;
							// Keep Busy=TRUE for paused commands, set Result to indicate interlock issue
							CommandStatus.Result := E_CommandResult.InterlockLost;
							IF (_iCommandConfiguration <> 0) THEN
								IF __ISVALIDREF(_iCommandConfiguration.P_CommandConfiguration.BaseConfiguration) THEN
									IF _iCommandConfiguration.P_CommandConfiguration.BaseConfiguration.LogTraceConfiguration.What.xLogToEventLogger AND NOT SUPER^.BaseStatus.LogTraceStatus.InterlockLossShown THEN
										TraceWithSeverity(Message := 'Command paused due to interlock loss (AbortOnInterlockDrop=FALSE)', Severity := Global.TcEventSeverity.Warning);
										SUPER^.BaseStatus.LogTraceStatus.InterlockLossShown := TRUE;
									END_IF
								END_IF
							ELSE
								// WARNING: Event logging disabled - configuration interface is null
								TraceWithSeverity(Message := 'WARNING: _iCommandConfiguration is null in _MonitorInterlocks - paused due to interlock loss logging disabled', Severity := Global.TcEventSeverity.Warning);
							END_IF
					END_IF
				END_IF
			END_IF
		END_IF
	END_IF
ELSE
	// CRITICAL: _iCommandConfiguration is null - cannot monitor interlocks or timeouts
	TraceWithSeverity(Message := 'CRITICAL: _iCommandConfiguration is null in _MonitorInterlocks - safety monitoring disabled', Severity := Global.TcEventSeverity.Error);
	RETURN;
END_IF
END_METHOD

METHOD PROTECTED _ProcessStateTransitions
// Policy B: Progress through states until reaching stable state (Monitor or Complete)
// This allows commands to complete within a single component cycle
REPEAT
    CASE CommandStatus.StepState OF
    E_CommandState.Idle:
        // Transition Idle → Execute when Busy flag is set (from Execute method)
        IF CommandStatus.BaseStatus.Busy AND CommandStatus.Result = E_CommandResult.Accepted THEN
            CommandStatus.StepState := E_CommandState.Execute;
            // Policy H: Increment try count on first transition into Execute (actual execution start)
            CommandStatus.CommandTryCount := CommandStatus.CommandTryCount + 1;

